ELSE
	bDone	:= FALSE;
END_IF

END_FUNCTION_BLOCK

// ---- POUs/METS/Common LIB/08_SOFTWARE LIB/Maths FBs/FB_CumulativeAverage.TcPOU
(* fAverage = sum of fInput samples / no of samples;  individual samples are not recorded *)
FUNCTION_BLOCK FB_CumulativeAverage
VAR_INPUT
	bEnable			: BOOL;		(* start cumulative calculation *)
	fInput			: LREAL;		(* input position *)
	tSamplePeriod	: TIME;		(* time period between each new value being logged *)
END_VAR
VAR_OUTPUT
	bRunning		: BOOL;		(* moving window being calculated without problem *)
	bNewValue		: BOOL;		(* set TRUE when a new value is logged and output is updated *)
	fAverage		: LREAL;	(* change in input value per second *)
	fMaxValue		: LREAL;	(* highest input value seen *)
	fMinValue		: LREAL;	(* lowest input value seen *)
END_VAR
VAR
	fbTaskTime		: FB_SYSTEM_TaskInfo;
	fTaskCycleTime	: LREAL;
	fbEnable		: R_TRIG;
	nLoggedSamples	: UDINT;
	fTimer			: LREAL;
	fSamplePeriod	: LREAL;
	fAccumulator	: LREAL;
END_VAR
(*
-------------------------------------------------------------------------------------------------
Date		Version	Author	Comments
-------------------------------------------------------------------------------------------------
30/01/2015	3.00.00	PB		LREAL now used in place of REAL

-------------------------------------------------------------------------------------------------
07/03/2012	1.09.00	PB		TaskTime calculated on rising edge of bEnable
05/02/2010	1.00.00	PB		Initial release

-------------------------------------------------------------------------------------------------
*)

(* detect rising edge of bEnable *)
fbEnable(CLK := bEnable);

(* generate average value *)
IF bEnable = TRUE THEN

	(* on rising edge of bEnable *)
	IF fbEnable.Q = TRUE THEN

		(* time base of current task *)
		fbTaskTime();
		fTaskCycleTime := fbTaskTime.fTaskTimeMicrosecs / 1000;

		fAccumulator := 0.0;
		nLoggedSamples := 0;
		fMaxValue := 0.0;
		fMinValue := 0.0;
	END_IF

	(* calculate sample period *)
	fSamplePeriod := MAX(fTaskCycleTime, TIME_TO_REAL(tSamplePeriod));

	(* update sample timer *)
	fTimer := fTimer + fTaskCycleTime;

	(* time to store new sample *)
	IF fTimer >= fSamplePeriod THEN

		(* set new value logged flag *)
		bNewValue := TRUE;

		(* update accumulator and samples and calculate new average *)
		fAccumulator := fAccumulator + fInput;
		nLoggedSamples := nLoggedSamples + 1;
		fAverage := F_SafeDIV(fAccumulator, UDINT_TO_REAL(nLoggedSamples));

		(* on 1st sample, set Max and Min Values = fInput *)
		IF nLoggedSamples = 1 THEN

			fMaxValue := fInput;
			fMinValue := fInput;
		END_IF

		(* update maximum and minimum values seen during average calculation *)
		fMaxValue := MAX(fInput, fMaxValue);
		fMinValue := MIN(fInput, fMinValue);

		(* remove complete sample time from timer *)
		fTimer := fTimer - fSamplePeriod;

	(* no new sample *)
	ELSE

		bNewValue := FALSE;
	END_IF

(* sampling disabled *)
ELSE

	bRunning := FALSE;
	bNewValue := FALSE;
	fAverage := fInput;
	nLoggedSamples := 0;
END_IF

END_FUNCTION_BLOCK

// ---- POUs/METS/Common LIB/08_SOFTWARE LIB/Maths FBs/FB_Interval.TcPOU
FUNCTION_BLOCK FB_Interval
(*
Version history:
Date		|	Version/Author 		|	Remark
----------------------------------------------------------------------------------------------------
04.07.12	|	2.000.001	PSA		|	Original Version
									|	Calculates the interval and ppm for 2 pulses.
*)
VAR_INPUT
	bSignal							: BOOL;						(* Input to detect the event *)
END_VAR
VAR_OUTPUT
	fInterval						: LREAL;					(* Gap between last 2 events  *)
	fPartsPerMinute					: LREAL;					(* Approximate parts per minute based on interval *)
END_VAR
VAR
	
	bInitOK 		: BOOL;
	fbTaskIndex		: GETCURTASKINDEX;
	
	fbSignalTrig					: R_TRIG;
	nCycleCount						: DWORD;
	nLastCycleCount					: DWORD;
END_VAR

fbSignalTrig(CLK := bSignal);

IF NOT bInitOK THEN
	(* get task indexc and task cycle time in seconds *)
	fbTaskIndex();
END_IF

bInitOK := fbTaskIndex.Index <> 0;

IF fbSignalTrig.Q AND bInitOK THEN
	
	nCycleCount :=  _TaskInfo[fbTaskIndex.Index].CycleCount;
	fInterval := DWORD_TO_LREAL(nCycleCount - nLastCycleCount) * (DWORD_TO_LREAL(_TaskInfo[fbTaskIndex.Index].CycleTime) / 10000000);
	nLastCycleCount :=  _TaskInfo[fbTaskIndex.Index].CycleCount;
	fPartsPerMinute := F_SafeDIV(60,fInterval);
END_IF

END_FUNCTION_BLOCK

// ---- POUs/METS/Common LIB/08_SOFTWARE LIB/Maths FBs/FB_MovingAverage.TcPOU
FUNCTION_BLOCK FB_MovingAverage
(*
Version history:
Date		|	Version/Author 		|	Remark
----------------------------------------------------------------------------------------------------
21.05.15	|	3.000.001	PSA		|	Original version
									|	Calculates a rolling average.
*)
VAR_INPUT
	bNewValue						: BOOL;						(* Input to detect the event *)
	bReset							: BOOL;						(* Resets the average value *)
	fLimit							: LREAL;					(* Limit value to inhibit bad data *)
END_VAR
VAR_OUTPUT
	nSamples						: DWORD := 1;
	fAverage						: LREAL := 0.0;
END_VAR
VAR
	fbTrig							: R_TRIG;
	fbResetTrig						: R_TRIG;
	FB_Interval1					: FB_Interval;
END_VAR

FB_Interval1(bSignal:= bNewValue);

fbTrig(CLK := bNewValue);
IF fbTrig.Q THEN
	IF FB_Interval1.fPartsPerMinute < fLimit THEN
		fAverage := ((fAverage * (nSamples - 1)) + FB_Interval1.fPartsPerMinute ) / nSamples;
		nSamples := nSamples + 1;
	END_IF
END_IF

fbResetTrig(CLK := bReset);
IF fbResetTrig.Q THEN
	nSamples := 1;
	fAverage := 0.0;
END_IF

END_FUNCTION_BLOCK

// ---- POUs/METS/Common LIB/08_SOFTWARE LIB/Maths FBs/FB_MovingAverageEvent.TcPOU
(* moving average over specified number if values logged on rising edge of bLogEvent *)
FUNCTION_BLOCK FB_MovingAverageEvent
VAR_INPUT
	bEnable			: BOOL;		(* set TRUE to enable moving average calculation.  fAverage = fInput when set FALSE *)
	bLogEvent		: BOOL;		(* log new value on FALSE-TRUE transition *)
	fInput			: LREAL;	(* input value *)
	nSamples		: UINT;		(* number of logged values to use *)
END_VAR
VAR_OUTPUT
	bRunning		: BOOL;		(* moving window being calculated without problem *)
	bError			: BOOL;		(* TRUE = nSamples is larger than size of internal array *)
	bNewValue		: BOOL;		(* set TRUE when a new value has been logged and fAverage updated *)
	fAverage		: LREAL;	(* moving average of last nSamples of fInput *)
	fMaxSample		: LREAL;	(* max value of samples being used *)
	fMinSample		: LREAL;	(* min value of samples being used *)
END_VAR
VAR
	fbEnable		: R_TRIG;
	arrValue		: ARRAY[1..120] OF LREAL;
	nMaxSamples		: UINT;
	fbLogEvent		: R_TRIG;
	nIndex			: UINT;
	nLoggedSamples	: UINT;
END_VAR
(*
-------------------------------------------------------------------------------------------------
Date		Version	Author	Comments
-------------------------------------------------------------------------------------------------
30/01/2015	3.00.00	PB		LREAL now used in place of REAL

-------------------------------------------------------------------------------------------------
07/03/2012	1.09.00	PB		MaxSamples is calculated and data array is cleared on rising edge of bEnable
05/02/2010	1.00.00	PB		Initial release

-------------------------------------------------------------------------------------------------
*)

(* detect rising edge of bEnable *)
fbEnable(CLK := bEnable);

(* log new value on rising edge of bExecute *)
fbLogEvent(CLK:= bLogEvent);

(* moving average enabled *)
IF bEnable = TRUE THEN

	(* on rising edge of bEnable *)
	IF fbEnable.Q = TRUE THEN

		(* clear array *)
		MEMSET(ADR(arrValue), 16#00, SIZEOF(arrValue));

		(* calculate max no of samples that can be handled *)
		nMaxSamples := SIZEOF(arrValue) / SIZEOF(arrValue[1]);
	END_IF

	(* no of samples specified exceeds size of array *)
	IF nSamples > nMaxSamples THEN

		(* set ERROR flag, use maximum number of samples allowed *)
		bError := TRUE;
		nSamples := nMaxSamples;
	END_IF

	(* log new value *)
	IF fbLogEvent.Q = TRUE THEN

		nLoggedSamples := MIN(nLoggedSamples + 1, nSamples);
		bNewValue := TRUE;

		(* shift data by 1 element in fValue and add new sample to fValue array *)
		MEMMOVE(ADR(arrValue[2]), ADR(arrValue[1]), SIZEOF(arrValue[1]) * (nMaxSamples - 1));
		arrValue[1] := fInput;

		(* calculate average value over specified period of time *)
		fAverage := 0.0;
		FOR nIndex := 1 TO nLoggedSamples DO

			(* add all sampled values *)
			fAverage := fAverage + arrValue[nIndex];

			(* new max sample or 1st value on scan *)
			IF arrValue[nIndex] > fMaxSample OR nIndex = 1 THEN

				fMaxSample := arrValue[nIndex];
			END_IF

			(* new min sample or 1st value on scan *)
			IF arrValue[nIndex] < fMinSample OR nIndex = 1 THEN

				fMinSample := arrValue[nIndex];
			END_IF
		END_FOR

		(* divide by number of samples used to return average value *)
		fAverage := F_SafeDIV(fAverage, UINT_TO_REAL(nLoggedSamples));

	(* no new value *)
	ELSE

		bNewValue := FALSE;
	END_IF

	bRunning := TRUE;

(* moving average disabled, output = input *)
ELSE

	bRunning := FALSE;
	bError := FALSE;
	bNewValue := FALSE;
	fAverage := fInput;
	nLoggedSamples := 0;
END_IF

END_FUNCTION_BLOCK

// ---- POUs/METS/Common LIB/08_SOFTWARE LIB/Maths FBs/FB_MovingAverageTimer.TcPOU
(* Returns a moving average over the last N cycles.  Values are taken on fixed timebase
and added to a buffer, new value replaces oldest value when 120 sample buffer is full. 
No of samples used for fAverage is calculated as tAveragePeriod / tSamplePeriod *)
FUNCTION_BLOCK FB_MovingAverageTimer
VAR_INPUT
	bEnable			: BOOL;		(* set TRUE to enable moving average calculation.  fAverage = fInput when set FALSE *)
	fInput			: LREAL;	(* input position *)
	tSamplePeriod	: TIME;		(* time period between each new value being logged, T#0ms = every cycle *)
	tAveragePeriod	: TIME;		(* time period over which to asses change of input value *)
END_VAR
VAR_OUTPUT
	bRunning		: BOOL;		(* moving window being calculated without problem *)
	bError			: BOOL;		(* error condition active *)
	bNewValue		: BOOL;		(* set TRUE when a new value is logged and output is updated *)
	fAverage		: LREAL;	(* change in input value per second *)
	fMaxSample		: LREAL;	(* max value of samples being used *)
	fMinSample		: LREAL;	(* min value of samples being used *)
END_VAR
VAR
	fbEnable		: R_TRIG;
	arrValue		: ARRAY[1..120] OF LREAL;
	fbTaskTime		: FB_SYSTEM_TaskInfo;
	fTaskCycleTime	: LREAL;
	nMaxSamples		: UINT;
	fSamplePeriod	: LREAL;
	fAveragePeriod	: LREAL;
	nSamples		: UINT;
	fTimer			: LREAL;
	nLoggedSamples	: UINT;
	nIndex			: UINT;
END_VAR
(*
-------------------------------------------------------------------------------------------------
Date		Version	Author	Comments
-------------------------------------------------------------------------------------------------
30/01/2015	3.00.00	PB		LREAL now used in place of REAL

-------------------------------------------------------------------------------------------------
07/03/2012	1.09.00	PB		TaskTime and MaxSamples are calculated and arrValue is cleared on rising edge of bEnable
05/02/2010	1.00.00	PB		Initial release

-------------------------------------------------------------------------------------------------
*)

(* detect rising edge of bEnable *)
fbEnable(CLK := bEnable);

(* moving average enabled *)
IF bEnable = TRUE THEN

	(* on rising edge of bEnable *)
	IF fbEnable.Q = TRUE THEN

		(* time base of current task *)
		fbTaskTime();
		fTaskCycleTime := fbTaskTime.fTaskTimeMicrosecs / 1000;

		(* clear array *)
		MEMSET(ADR(arrValue), 16#00, SIZEOF(arrValue));

		(* calculate max no of samples that can be handled *)
		nMaxSamples := SIZEOF(arrValue) / SIZEOF(arrValue[1]);
	END_IF

	(* calculate internal values required *)
	fSamplePeriod := MAX(fTaskCycleTime, TIME_TO_REAL(tSamplePeriod));
	fAveragePeriod := MAX(fTaskCycleTime, TIME_TO_REAL(tAveragePeriod));
	nSamples := lREAL_TO_UINT(F_SafeDIV(fAveragePeriod, fSamplePeriod));

	(* no of samples specified exceeds size of array *)
	IF nSamples > nMaxSamples THEN

		(* set ERROR flag, use maximum number of samples allowed *)
		bError := TRUE;
		nSamples := nMaxSamples;
	END_IF

	(* update timer *)
	fTimer := fTimer + fTaskCycleTime;

	(* time to store new sample *)
	IF fTimer >= fSamplePeriod THEN

		bNewValue := TRUE;
		nLoggedSamples := MIN(nLoggedSamples + 1, nSamples);

		(* shift data by 1 element in fValue and add new sample to array *)
		MEMMOVE(ADR(arrValue[2]), ADR(arrValue[1]), SIZEOF(arrValue[1]) * (nMaxSamples - 1));
		arrValue[1] := fInput;

		(* remove complete sample time from timer *)
		fTimer := fTimer - fSamplePeriod;

		(* calculate average value over specified period of time *)
		fAverage := 0.0;
		FOR nIndex := 1 TO nLoggedSamples DO

			(* add all sampled values *)
			fAverage := fAverage + arrValue[nIndex];

			(* new max sample or 1st value on scan *)
			IF arrValue[nIndex] > fMaxSample OR nIndex = 1 THEN

				fMaxSample := arrValue[nIndex];
			END_IF

			(* new min sample or 1st value on scan *)
			IF arrValue[nIndex] < fMinSample OR nIndex = 1 THEN

				fMinSample := arrValue[nIndex];
			END_IF
		END_FOR

		(* divide by number of samples used to return average value *)
		fAverage := F_SafeDIV(fAverage, UINT_TO_REAL(nLoggedSamples));

	(* no new sample *)
	ELSE

		bNewValue := FALSE;
	END_IF

	bRunning := TRUE;

(* moving average disabled *)
ELSE

	bRunning := FALSE;
	bError := FALSE;
	bNewValue := FALSE;
	fAverage := fInput;
	nLoggedSamples := 0;
END_IF

END_FUNCTION_BLOCK

// ---- POUs/METS/Common LIB/08_SOFTWARE LIB/Maths FBs/FB_MovingWindowEvent.TcPOU
(* Returns the difference between new value and historical value.
Values are added to a buffer on rising edge of bLogEvent, oldest value is deleted after 120 samples.
No of samples to be used is specified by nSamples *)
FUNCTION_BLOCK FB_MovingWindowEvent
VAR_INPUT
	bEnable			: BOOL;
	bLogEvent		: BOOL;		(* log new input value and time *)
	fInput			: LREAL;	(* input value *)
	fTime			: LREAL;	(* time in secs *)
	nSamples		: UINT;		(* number of events to log *)
END_VAR
VAR_OUTPUT
	bRunning		: BOOL;		(* moving window being calculated without problem *)
	bError			: BOOL;		(* error condition active *)
	bNewValue		: BOOL;		(* set TRUE when a new value is logged and output is updated *)
	fDeltaPerSec	: LREAL;	(* change in input value per second *)
	fDeltaPerMin	: LREAL;	(* change in input value per minute *)
	fDeltaPerHour	: LREAL;	(* change in input value per hour *)
END_VAR
VAR
	fbEnable		: R_TRIG;
	arrValue		: ARRAY[1..120] OF LREAL;
	arrTime			: ARRAY[1..120] OF LREAL;
	nMaxSamples		: UINT;
	nLoggedSamples	: UINT;
	fbLogEvent		: R_TRIG;
END_VAR
(*
-------------------------------------------------------------------------------------------------
Date		Version	Author	Comments
-------------------------------------------------------------------------------------------------
30/01/2015	3.00.00	PB		LREAL now used in place of REAL

-------------------------------------------------------------------------------------------------
07/03/2012	1.09.00	PB		MaxSamples is calculated and data arrays are cleared on rising edge of bEnable
05/02/2010	1.00.00	PB		Initial release

-------------------------------------------------------------------------------------------------
*)

(* detect rising edge of bEnable *)
fbEnable(CLK := bEnable);

(* check for rising edge on bLogEvent input *)
fbLogEvent(CLK:= bLogEvent);

(* moving window enabled *)
IF bEnable = TRUE THEN

	(* on rising edge of bEnable *)
	IF fbEnable.Q = TRUE THEN

		(* clear arrays *)
		MEMSET(ADR(arrValue), 16#00, SIZEOF(arrValue));
		MEMSET(ADR(arrTime), 16#00, SIZEOF(arrTime));

		(* calculate max no of samples that can be handled *)
		nMaxSamples := SIZEOF(arrValue) / SIZEOF(arrValue[1]);
	END_IF

	(* no of samples specified exceeds size of array *)
	IF nSamples > nMaxSamples THEN

		(* set ERROR flag, use maximum number of samples allowed *)
		bError := TRUE;
		nSamples := nMaxSamples;
	END_IF

	(* log new value *)
	IF fbLogEvent.Q = TRUE THEN

		bNewValue := TRUE;
		nLoggedSamples := MIN(nLoggedSamples + 1, nSamples);

		(* shift data by 1 element in fArray and add new sample to array *)
		MEMMOVE(ADR(arrValue[2]), ADR(arrValue[1]), SIZEOF(arrValue[1]) * (nMaxSamples - 1));
		MEMMOVE(ADR(arrTime[2]), ADR(arrTime[1]), SIZEOF(arrTime[1]) * (nMaxSamples - 1));
		arrValue[1] := fInput;
		arrTime[1] := fTime;

		(* need 2 samples before change of input over time can be calculated *)
		IF nLoggedSamples > 1 THEN

			(* calculate change of input over change of time *)
			fDeltaPerSec := F_SafeDIV((arrValue[1] - arrValue[nLoggedSamples]), (arrTime[1] - arrTime[nLoggedSamples]));
			fDeltaPerMin := fDeltaPerSec * 60.0;
			fDeltaPerHour := fDeltaPerMin * 60.0;
		END_IF

	(* no new sample *)
	ELSE

		bNewValue := FALSE;
	END_IF

(* moving window disabled *)
ELSE

	bRunning := FALSE;
	bError := FALSE;
	bNewValue := FALSE;
	fDeltaPerSec := 0.0;
	fDeltaPerMin := 0.0;
	nLoggedSamples := 0;
END_IF

END_FUNCTION_BLOCK

// ---- POUs/METS/Common LIB/08_SOFTWARE LIB/Maths FBs/FB_MovingWindowTimer.TcPOU
(* Returns the difference between new value and historical value.
Values are added to a buffer on a fixed timebase, oldest value is deleted after 120 samples.
Time difference between assessed values is specified by tWindowPeriod *)
FUNCTION_BLOCK FB_MovingWindowTimer
VAR_INPUT
	bEnable			: BOOL;
	fInput			: LREAL;	(* input position *)
	tSamplePeriod	: TIME;		(* time period between each new value being logged, T#0ms = every cycle *)
	tWindowPeriod	: TIME;		(* time period over which to asses change of input value *)
END_VAR
VAR_OUTPUT
	bRunning		: BOOL;		(* moving window being calculated without problem *)
	bError			: BOOL;		(* error condition active *)
	bNewValue		: BOOL;		(* set TRUE when a new value is logged and output is updated *)
	fDeltaPerSec	: LREAL;	(* change in input value per second *)
	fDeltaPerMin	: LREAL;	(* change in input value per minute *)
	fDeltaPerHour	: LREAL;	(* change in input value per hour *)
END_VAR
VAR
	fbEnable		: R_TRIG;
	fbTaskTime		: FB_SYSTEM_TaskInfo;
	fTaskCycleTime	: LREAL;
	arrValue		: ARRAY[1..120] OF LREAL;
	nMaxSamples		: UINT;
	fSamplePeriod	: LREAL;
	fWindowPeriod	: LREAL;
	nSamples		: UINT;
	fTimer			: LREAL;
	nLoggedSamples	: UINT;
END_VAR
(*
-------------------------------------------------------------------------------------------------
Date		Version	Author	Comments
-------------------------------------------------------------------------------------------------
30/01/2015	3.00.00	PB		LREAL now used in place of REAL

-------------------------------------------------------------------------------------------------
07/03/2012	1.09.00	PB		TaskTime and MaxSamples are calculated and arrValue is cleared on rising edge of bEnable
05/02/2010	1.00.00	PB		Initial release

-------------------------------------------------------------------------------------------------
*)

(* detect rising edge of bEnable *)
fbEnable(CLK := bEnable);

(* moving window enabled *)
IF bEnable = TRUE THEN

	(* on rising edge of bEnable *)
	IF fbEnable.Q = TRUE THEN

		(* time base of current task *)
		fbTaskTime();
		fTaskCycleTime := fbTaskTime.fTaskTimeMicrosecs / 1000;

		(* clear array *)
		MEMSET(ADR(arrValue), 16#00, SIZEOF(arrValue));

		(* calculate max no of samples that can be handled *)
		nMaxSamples := SIZEOF(arrValue) / SIZEOF(arrValue[1]);
	END_IF

	fSamplePeriod := MAX(fTaskCycleTime, TIME_TO_REAL(tSamplePeriod));
	fWindowPeriod := MAX(fTaskCycleTime, TIME_TO_REAL(tWindowPeriod));
	nSamples := lREAL_TO_UINT(F_SafeDIV(fWindowPeriod, fSamplePeriod));

	(* no of samples specified exceeds size of array *)
	IF nSamples > nMaxSamples THEN

		(* set ERROR flag, use maximum number of samples allowed *)
		bError := TRUE;
		nSamples := nMaxSamples;
	END_IF

	(* update timer *)
	fTimer := fTimer + fTaskCycleTime;

	(* time to store new sample *)
	IF fTimer >= fSamplePeriod THEN

		bNewValue := TRUE;
		nLoggedSamples := MIN(nLoggedSamples + 1, nSamples);

		(* shift data by 1 element in fArray and add new sample to array *)
		MEMMOVE(ADR(arrValue[2]), ADR(arrValue[1]), SIZEOF(arrValue[1]) * (nMaxSamples - 1));
		arrValue[1] := fInput;

		(* remove complete sample time from timer *)
		fTimer := fTimer - fSamplePeriod;

		(* calculate position change over specified number of samples *)
		fDeltaPerSec := F_SafeDIV((arrValue[1] - arrValue[nLoggedSamples]) * 1000.0, (fSamplePeriod * UINT_TO_REAL(nLoggedSamples)));
		fDeltaPerMin := fDeltaPerSec * 60.0;
		fDeltaPerHour := fDeltaPerMin * 60.0;

	(* no new sample *)
	ELSE

		bNewValue := FALSE;
	END_IF

(* moving window disabled *)
ELSE

	bRunning := FALSE;
	bError := FALSE;
	bNewValue := FALSE;
	fDeltaPerSec := 0.0;
	fDeltaPerMin := 0.0;
	nLoggedSamples := 0;
END_IF

END_FUNCTION_BLOCK

// ---- POUs/METS/Common LIB/08_SOFTWARE LIB/Maths FBs/F_ApplyTimeOffset.TcPOU
(* apply specified TIME offset to TIMESTRUCT value *)
FUNCTION F_ApplyTimeOffset : TIMESTRUCT
VAR_INPUT
	sTime			: TIMESTRUCT;	(* system time *)
	nTimeOffset		: DINT;			(* offset time, specified in ms *)
END_VAR
VAR
	nFileTime		: T_ULARGE_INTEGER;
END_VAR
(*
-------------------------------------------------------------------------------------------------
Date		Version	Author	Comments
-------------------------------------------------------------------------------------------------
30/01/2015	3.00.00	PB		Moved from Sewtec_CaseTrace.lib

-------------------------------------------------------------------------------------------------
03/08/2012	1.39.00	PB		Initial release

-------------------------------------------------------------------------------------------------
*)

(* offset time is specified *)
IF nTimeOffset <> 0 THEN

	(* convert TIMESTRUCT to T_ULARGE_INTEGER via T_FILETIME *)
	nFileTime := F_FileTimeToULarge(SYSTEMTIME_TO_FILETIME(sTime));

	(* positive time offset *)
	IF nTimeOffset >= 0 THEN

		(* convert DINT (1 = 1ms) to T_ULARGE_INTEGER (1 = 100ns) and add to system time *)
		nFileTime := UInt64Add64(nFileTime, UInt32x32To64(ABS(DINT_TO_DWORD(nTimeOffset)), 10000));

	(* negative time offset *)
	ELSE

		(* convert DINT (1 = 1ms) to T_ULARGE_INTEGER (1 = 100ns) and subtract from system time *)
		nFileTime := UInt64Sub64(nFileTime, UInt32x32To64(ABS(DINT_TO_DWORD(nTimeOffset)), 10000));
	END_IF

	(* convert T_ULARGE_INTEGER to TIMESTRUCT (via T_FILETIME *)
	F_ApplyTimeOffset := FILETIME_TO_SYSTEMTIME(F_ULargeToFileTime(nFileTime));

(* offset time = 0 *)
ELSE

	(* set Offset Time = System Time *)
	F_ApplyTimeOffset := sTime;
END_IF

END_FUNCTION

// ---- POUs/METS/Common LIB/08_SOFTWARE LIB/Maths FBs/F_ULargeToFileTime.TcPOU
(* convert value from 64-bit T_ULARGE_INTEGER to 64-bit T_FILETIME *)
FUNCTION F_ULargeToFileTime : T_FILETIME
VAR_INPUT
	nULarge			: T_ULARGE_INTEGER;
END_VAR
VAR
END_VAR
(*
-------------------------------------------------------------------------------------------------
Date		Version	Author	Comments
-------------------------------------------------------------------------------------------------
30/01/2015	3.00.00	PB		Moved from Sewtec_CaseTrace.lib

-------------------------------------------------------------------------------------------------
03/08/2012	1.39.00	PB		Initial release

-------------------------------------------------------------------------------------------------
*)

MEMMOVE(ADR(F_ULargeToFileTime), ADR(nULarge), SIZEOF(F_ULargeToFileTime));

END_FUNCTION

// ---- POUs/METS/Common LIB/08_SOFTWARE LIB/Maths FBs/F_CompareSign.TcPOU
(* F_CompareSign compares the sign of 2 LREAL values and gives TRUE if both values *)
(* are non-zero and have opposite sign *)
FUNCTION F_CompareSign : BOOL
VAR_INPUT
	fValue1		: LREAL;
	fValue2		: LREAL;
END_VAR
VAR
END_VAR
(*
-------------------------------------------------------------------------------------------------
Date		Version	Author	Comments
-------------------------------------------------------------------------------------------------
30/01/2015	3.00.00	PB		No change

-------------------------------------------------------------------------------------------------
05/02/10	1.00.00	PB		Initial release

-------------------------------------------------------------------------------------------------
*)

(* input values are both non-zero *)
IF fValue1 <> 0.0 AND fValue2 <> 0.0 THEN

	(* values have different signs *)
	IF F_GetSign(fValue1) <> F_GetSign(fValue2) THEN

		F_CompareSign := TRUE;

	(* values have same sign *)
	ELSE

		F_CompareSign := FALSE;
	END_IF

(* one of input values is zero *)
ELSE

	F_CompareSign := FALSE;
END_IF

END_FUNCTION

// ---- POUs/METS/Common LIB/08_SOFTWARE LIB/Maths FBs/F_GetSign.TcPOU
(* F_GetSign indicates the sign of the input LREAL value, set to 0 is input value is 0 *)
(* 1 = +ive, -1 = -ive *)
FUNCTION F_GetSign : INT
VAR_INPUT
	fValue		: LREAL;
END_VAR
VAR
END_VAR
(*
-------------------------------------------------------------------------------------------------
Date		Version	Author	Comments
-------------------------------------------------------------------------------------------------
30/01/2015	3.00.00	PB		No change

-------------------------------------------------------------------------------------------------
05/02/10	1.00.00	PB		Initial release

-------------------------------------------------------------------------------------------------
*)

(* input value is positive *)
IF fValue > 0.0 THEN

	F_GetSign := 1;

(* input value is negative *)
ELSIF fValue < 0.0 THEN

	F_GetSign := -1;

(* input value is zero *)
ELSE

	F_GetSign := 0;
END_IF

END_FUNCTION

// ---- POUs/METS/Common LIB/08_SOFTWARE LIB/Maths FBs/F_Interpolate.TcPOU
(* linear interpolation between 2 specified points (X,Y) using y=mx+c *)
FUNCTION F_Interpolate : LREAL
VAR_INPUT
	fX1			: LREAL;	(* X for defined point 1 *)
	fY1			: LREAL;	(* Y for defined point 1 *)
	fX2			: LREAL;	(* X for defined point 2 *)
	fY2			: LREAL;	(* Y for defined point 2 *)
	fCurrX		: LREAL;	(* current X value *)
END_VAR
VAR
END_VAR
(*
-------------------------------------------------------------------------------------------------
Date		Version	Author	Comments
-------------------------------------------------------------------------------------------------
30/01/2015	3.00.00	PB		Initial release

-------------------------------------------------------------------------------------------------
*)

(* X values are identical *)
IF fX2 = fX1 THEN

	(* graph is a vertical line and cannot interpolate, output is fixed *)
	F_Interpolate := fX1;

(* X values are different *)
ELSE

	(* apply linear interpolation *)
	F_Interpolate := (((fY2 - fY1) * (fCurrX - fX1)) / (fX2 - fX1)) + fY1;
END_IF

END_FUNCTION

// ---- POUs/METS/Common LIB/08_SOFTWARE LIB/Maths FBs/F_ModuloPos.TcPOU
(* converts absolute position to modulo position, 0 <= fModuloPos < fModuloFactor *)
FUNCTION F_ModuloPos : LREAL
VAR_INPUT
	fAbsPos			: LREAL;	(* absolute position *)
	fModuloFactor	: LREAL;	(* modulo factor *)
END_VAR
VAR
END_VAR
(*
-------------------------------------------------------------------------------------------------
Date		Version	Author	Comments
-------------------------------------------------------------------------------------------------
30/01/2015	3.00.00	PB		Initial release

-------------------------------------------------------------------------------------------------
*)

(* absolute position is +ive *)
IF fAbsPos >= 0 THEN

	(* LMOD produces modulo position *)
	F_ModuloPos := LMOD(fAbsPos, fModuloFactor);

(* absolute position is -ive *)
ELSE

	(* LMOD gives negative value, add fModuloFactor to convert to positive value *)
	F_ModuloPos := LMOD(fAbsPos, fModuloFactor) + fModuloFactor;
END_IF

END_FUNCTION

// ---- POUs/METS/Common LIB/08_SOFTWARE LIB/Memory FBs/FB_StructureMonitor.TcPOU
(* monitor memory area for change of data, max 64Kbytes *)
FUNCTION_BLOCK FB_StructureMonitor
VAR_INPUT
	bEnable			: BOOL;		(* set TRUE to enable monitoring *)
	pSourceData		: POINTER TO BYTE;	(* pointer to source data *)
	nSourceBytes	: UDINT;	(* no of data bytes *)
	tUpdateTime		: TIME;		(* update time *)
END_VAR
VAR_OUTPUT
	bDataChanged	: BOOL;		(* TRUE = data changed *)
	nTotalChanges	: UDINT;	(* total number of memory changes detected *)
END_VAR
VAR

	nCurrentCheckSum	: WORD;
	nLastCheckSum	: WORD;
	fbUpdateTimer		: FB_PulseGenerator;
END_VAR

(* update timer *)
fbUpdateTimer(
	bEnable		:= bEnable,
	tPeriod		:= tUpdateTime
);

(* data not changed on last pass *)
IF bDataChanged = FALSE THEN

	(* check for change of data *)
	IF fbUpdateTimer.bOutput = TRUE THEN

		nCurrentCheckSum := F_Checksum_CRC16(bEnable	:= bEnable, pSrcAddr := pSourceData, nBytes := nSourceBytes, nStartCRC := 16#FFFF);

		IF nCurrentCheckSum <> nLastCheckSum THEN

			nTotalChanges := nTotalChanges + 1;
			bDataChanged := TRUE;
		END_IF
	END_IF

(* data change detected on last pass *)
ELSE
	nLastCheckSum := nCurrentCheckSum;
	bDataChanged := FALSE;
END_IF

END_FUNCTION_BLOCK

// ---- POUs/METS/Common LIB/08_SOFTWARE LIB/Memory FBs/F_Checksum_CRC16.TcPOU
(* calculate 16-bit checksum on a memory area *)
FUNCTION F_Checksum_CRC16 : WORD
VAR_INPUT
	bEnable		: BOOL;				(* TRUE = calculate checksum *)
	pSrcAddr	: POINTER TO BYTE;	(* pointer to 1st byte of memory area *)
	nBytes		: UDINT;			(* no of bytes to be included in checksum calculation *)
	nStartCRC	: UINT;				(* initial value used for checksum calculation *)
END_VAR
VAR
END_VAR
(*
-------------------------------------------------------------------------------------------------
Date		Version	Author	Comments
-------------------------------------------------------------------------------------------------
30/01/2015	3.00.00	PB		No change

-------------------------------------------------------------------------------------------------
05/02/10	1.00.00	PB		Initial release

-------------------------------------------------------------------------------------------------
*)

(* calculate checksum when bEnable = TRUE *)
IF bEnable = TRUE THEN

	F_Checksum_CRC16 := F_DATA_TO_CRC16_CCITT(pSrcAddr, nBytes, nStartCRC);
END_IF

END_FUNCTION

// ---- POUs/METS/Common LIB/08_SOFTWARE LIB/Memory FBs/F_8BitsToByte.TcPOU
(* moves 8 bits into a single byte *)
FUNCTION F_8BitsToByte : BYTE
VAR_INPUT
	bInput1		: BOOL;
	bInput2		: BOOL;
	bInput3		: BOOL;
	bInput4		: BOOL;
	bInput5		: BOOL;
	bInput6		: BOOL;
	bInput7		: BOOL;
	bInput8		: BOOL;
END_VAR
VAR
END_VAR
(*
-------------------------------------------------------------------------------------------------
Date		Version	Author	Comments
-------------------------------------------------------------------------------------------------
30/01/2015	3.00.00	PB		Initial release

-------------------------------------------------------------------------------------------------
*)

F_8BitsToByte.0 := bInput1;
F_8BitsToByte.1 := bInput2;
F_8BitsToByte.2 := bInput3;
F_8BitsToByte.3 := bInput4;
F_8BitsToByte.4 := bInput5;
F_8BitsToByte.5 := bInput6;
F_8BitsToByte.6 := bInput7;
F_8BitsToByte.7 := bInput8;

END_FUNCTION

// ---- POUs/METS/Common LIB/08_SOFTWARE LIB/Memory FBs/F_GetBitState.TcPOU
(* returns status of specified bit from a DWORD value *)
FUNCTION F_GetBitState : BOOL
VAR_INPUT
	bEnable		: BOOL;		(* set TRUE to update output with state of target bit in nValue *)
	nTargetBit	: BYTE;		(* number of bit in nValue to be returned (0-31) *)
	nValue		: DWORD;	(* value from which target bit should be extracted *)
END_VAR
VAR
	nMaskValue	: DWORD;
END_VAR
(*
-------------------------------------------------------------------------------------------------
Date		Version	Author	Comments
-------------------------------------------------------------------------------------------------
30/01/2015	3.00.00	PB		No change

-------------------------------------------------------------------------------------------------
21/05/2010	1.03.00	PB		Initial release

-------------------------------------------------------------------------------------------------
*)

(* bit evaluation is enabled *)
IF bEnable = TRUE THEN

	(* target bit must be 0-31 *)
	IF nTargetBit <= 31 THEN

		(* calculate mask value from specified target bit *)
		nMaskValue := lREAL_TO_DWORD(EXPT(2, nTargetBit));

		(* compare nDWord AND nMaskValue, target bit is TRUE if value > 0 *)
		IF (nValue AND nMaskValue) > 0 THEN

			F_GetBitState := TRUE;

		(* target bit is FALSE *)
		ELSE

			F_GetBitState := FALSE;
		END_IF

	(* target bit out of range *)
	ELSE

		F_GetBitState := FALSE;
	END_IF

(* bit evaluation disabled *)
ELSE

	F_GetBitState := FALSE;
END_IF

END_FUNCTION

// ---- POUs/METS/Common LIB/08_SOFTWARE LIB/Memory FBs/F_PointerToByteADD.TcPOU
(* add offset to POINTER TO BYTE value *)
FUNCTION F_PointerToByteADD : PVOID
VAR_INPUT
	pPointer		: PVOID;	(* base pointer *)
	nOffset			: UDINT;			(* pointer offset *)
END_VAR
VAR
	nPointer		: ULINT;
	nPointerOffset	: ULINT;
END_VAR
(*
-------------------------------------------------------------------------------------------------
Date		Version	Author	Comments
-------------------------------------------------------------------------------------------------
30/01/2015	3.00.00	PB		No change

-------------------------------------------------------------------------------------------------
05/02/10	1.00.00	PB		Initial release

-------------------------------------------------------------------------------------------------
*)

nPointer := pPointer;					(* convert pointer to UDINT *)
nPointerOffset := nPointer + nOffset;	(* add offset *)
F_PointerToByteADD := nPointerOffset;	(* convert UDINT back to pointer *)

END_FUNCTION

// ---- POUs/METS/Common LIB/08_SOFTWARE LIB/Memory FBs/F_PointerToWordADD.TcPOU
(* add offset to POINTER TO WORD value *)
FUNCTION F_PointerToWordADD : PVOID
VAR_INPUT
	pPointer		: PVOID;	(* base pointer *)
	nOffset			: UDINT;			(* pointer offset *)
END_VAR
VAR
	nPointer		: ULINT;
	nPointerOffset	: ULINT;
END_VAR
(*
-------------------------------------------------------------------------------------------------
Date		Version	Author	Comments
-------------------------------------------------------------------------------------------------
30/01/2015	3.00.00	PB		No change

-------------------------------------------------------------------------------------------------
05/02/10	1.00.00	PB		Initial release

-------------------------------------------------------------------------------------------------
*)

nPointer := pPointer;					(* convert pointer to UDINT *)
nPointerOffset := nPointer + nOffset;	(* add offset *)
F_PointerToWordADD := nPointerOffset;	(* convert UDINT back to pointer *)

END_FUNCTION

// ---- POUs/METS/Common LIB/08_SOFTWARE LIB/Memory FBs/F_SetBitState.TcPOU
(* updates state of specified bit in nDWord value *)
FUNCTION F_SetBitState : DWORD
VAR_INPUT
	bEnable		: BOOL;		(* set TRUE to update state of target bit in nValue *)
	nTargetBit	: BYTE;		(* bit number of bit to be updated (0-31) *)
	nSetState	: BOOL;		(* state to which nTargetBit should be set *)
END_VAR

VAR
	nMaskValue	: DWORD;
END_VAR
(*
-------------------------------------------------------------------------------------------------
Date		Version	Author	Comments
-------------------------------------------------------------------------------------------------
30/01/2015	3.00.00	PB		No change

-------------------------------------------------------------------------------------------------
26/05/2010	1.03.01	PB		nValue now updated as well as F_SetBitState
21/05/2010	1.03.00	PB		Initial release

-------------------------------------------------------------------------------------------------
*)
(*All VAR_IN_OUT variables have been moved to the end of the declaration due to compatibility reasons*)
VAR_IN_OUT
	nValue		: DWORD;	(* value in which target bit should be updated *)
END_VAR

(* bit update is enabled *)
IF bEnable = TRUE THEN

	(* target bit must be 0-31 *)
	IF nTargetBit <= 31 THEN

		(* calculate mask value from specified target bit *)
		nMaskValue := LREAL_TO_DWORD(EXPT(2, nTargetBit));

		nValue := (nValue AND NOT nMaskValue) + (BOOL_TO_DWORD(nSetState) * nMaskValue);

	(* target bit out of range *)
	ELSE

		nValue := nValue;
	END_IF

(* bit update disabled *)
ELSE

	nValue := nValue;
END_IF

F_SetBitState := nValue;

END_FUNCTION

// ---- POUs/METS/Common LIB/08_SOFTWARE LIB/String FBs/FB_ExtractLongString.TcPOU
(* extracts a sub-string defined by prefix and suffix *)
FUNCTION_BLOCK FB_ExtractLongString
VAR_INPUT
	bExtractData		: BOOL;			(* set TRUE to remove prefix and suffix from strData *)
	nExtractChars		: UINT;			(* if suffix is blank, number of data chars to extract *)
	strPrefix			: T_MaxString;	(* prefix string *)
	strSuffix			: T_MaxString;	(* suffix string *)
END_VAR
VAR_IN_OUT
	strString			: T_LongSTRING;	(* string to be searched *)
END_VAR
VAR_OUTPUT
	bStringFound		: BOOL;			(* TRUE = sub-string with matching prefix/suffix found *)
	nStartPos			: UINT;			(* start pos of extracted string in strString *)
	strData				: T_LongSTRING;	(* extracted data *)
END_VAR
VAR
	nStringLen			: UINT;
	nPrefixLen			: UINT;
	nSuffixLen			: UINT;
	nEndPos				: UINT;
	bStartPosFound		: BOOL;
	bEndPosFound		: BOOL;
	nChars				: UINT;
	nMaxIndex			: UINT;
	nIndex				: UINT;

END_VAR
(*
-------------------------------------------------------------------------------------------------
DATE		Version	Author	Comments
-------------------------------------------------------------------------------------------------
30/01/2015	3.00.00	PB		Initial release

-------------------------------------------------------------------------------------------------
*)

(* calc string lengths *)
nStringLen := UDINT_TO_UINT(LEN2(ADR(strString)));
nPrefixLen := INT_TO_UINT(LEN(strPrefix));
nSuffixLen := INT_TO_UINT(LEN(strSuffix));

(* string to be searched is not empty and prefix or suffix or no or chars to extract is defined *)
IF nStringLen > 0 AND (nPrefixLen > 0 OR nSuffixLen > 0 OR nExtractChars > 0) THEN

	(* clear outputs *)
	bStringFound := FALSE;
	nChars := 0;
	nStartPos := 0;
	strData := '';

	(* initialise char index values *)
	bStartPosFound := FALSE;
	bEndPosFound := FALSE;
	nEndPos := 0;

	(* max search index, based on string length - 1 due to starting at 0 and length of prefix *)
	nMaxIndex := (nStringLen - 1) + (nPrefixLen - 1);

	(* for each character in the string *)
	FOR nIndex := 0 TO nMaxIndex DO

		(*IF nIndex = nMaxIndex  AND NOT bStartPosFound THEN

			strString :='1';

		(* prefix has not been found *)
		ELS*)IF bStartPosFound = FALSE THEN

			(* no prefix defined  *)
			IF nPrefixLen = 0 THEN

				(* start at beginning if string *)
				nStartPos := 1;
				bStartPosFound := TRUE;

			(* prefix defined  *)
			ELSE

				(* compare partial string with prefix *)
				IF MEMCMP(ADR(strString) + nIndex, ADR(strPrefix), nPrefixLen) = 0 THEN

					(* prefix position found *)
					nStartPos := nIndex + 1;
					bStartPosFound := TRUE;

					(* skip to end of prefix to continue search *)
					nIndex := nIndex + nPrefixLen - 1;
				END_IF
			END_IF

		(* suffix has not been found *)
		ELSIF bEndPosFound = FALSE THEN

			(* no suffix defined  *)
			IF nSuffixLen = 0 THEN

				(* start at 1st char of string *)
				bEndPosFound := TRUE;

				(* calculate end position *)
				nEndPos := MIN((nStartPos - 1) + nExtractChars + nPrefixLen, nStringLen);

			(* suffix defined  *)
			ELSE

				(* compare partial string with suffix *)
				IF MEMCMP(ADR(strString) + nIndex, ADR(strSuffix), nSuffixLen) = 0 THEN

					(* suffix position found, calculate end position *)
					nEndPos := nIndex + nSuffixLen;
					bEndPosFound := TRUE;

					(* no prefix defined and number of chars to extract is defined *)
					IF nPrefixLen = 0 AND nExtractChars > 0 THEN

						(* re-calculate start position *)
						nStartPos := MAX(nEndPos - nExtractChars - 1, 1);
					END_IF

					(* search complete, quit FOR loop *)
					EXIT;
				END_IF
			END_IF

		(* prefix and suffix found *)
		ELSE

			(* quit FOR loop *)
			EXIT;
		END_IF
	END_FOR

	(* start and end positions known *)
	IF bStartPosFound = TRUE AND bEndPosFound = TRUE THEN

		(* string has been found *)
		bStringFound := TRUE;

		(* return string without prefix and suffix *)
		IF bExtractData = TRUE THEN

			(* total chars to be moved to strData *)
			nChars := (nEndPos - (nStartPos - 1)) - nPrefixLen - nSuffixLen;

			(* 1 or more chars to be moved *)
			IF nChars > 0 THEN

				(* move data to strData *)
				MEMMOVE(ADR(strData), ADR(strString) + (nStartPos - 1) + nPrefixLen, nChars);
			END_IF

		(* return string with prefix and suffix *)
		ELSE

			(* total chars to be moved to strData *)
			nChars := nEndPos - (nStartPos - 1);

			(* 1 or more chars to be moved *)
			IF nChars > 0 THEN

				(* move data to strData *)
				MEMMOVE(ADR(strData), ADR(strString) + (nStartPos - 1), nChars);
			END_IF
		END_IF

		(* terminate strData *)
		MEMSET(ADR(strData) + nChars, 16#00, 1);

		(* 1 or more chars after strSuffix *)
		IF nStringLen > (nEndPos - (nStartPos - 1)) THEN

			(* shift post-suffix chars to prefix position *)
			MEMMOVE(ADR(strString) + (nStartPos - 1), ADR(strString) + nEndPos, nStringLen - (nEndPos - (nStartPos - 1)));
		END_IF

		(* terminate strString *)
		MEMSET(ADR(strString) + nStringLen - (nEndPos - (nStartPos - 1)), 16#00, 1);
	END_IF

(* string to be searched is empty or prefix and suffix and both blank *)
ELSE

	(* clear outputs *)
	bStringFound := FALSE;
	nChars := 0;
	strData := '';
END_IF

END_FUNCTION_BLOCK

// ---- POUs/METS/Common LIB/08_SOFTWARE LIB/String FBs/FB_ExtractString_v2.TcPOU
(* extracts a sub-string defined by prefix and suffix *)
FUNCTION_BLOCK FB_ExtractString_v2
VAR_INPUT
	bIgnoreCase		: BOOL;
	strPrefix		: STRING(10);	(* prefix string *)
	strSuffix		: STRING(10);	(* suffix string *)
	nExtractChars	: BYTE;			(* if suffix is blank, >0 = no of chars to extract , 0 = remainder of string *)
END_VAR
VAR_IN_OUT
	strString		: T_MaxString;	(* string to be searched *)
END_VAR
VAR_OUTPUT
	bStringFound	: BOOL;			(* TRUE = sub-string with matching prefix/suffix found *)
	nChars			: INT;			(* no of chars in sub-string *)
	strResult		: T_MaxString;	(* sub-string with prefix and suffix *)
END_VAR
VAR
	nPrefixPos		: INT;
	nSuffixPos		: INT;
	nIndex			: INT;
	strStringInt	: T_MaxString;
	strPrefixInt	: STRING(10);
	strSuffixInt	: STRING(10);
	strCheckString	: STRING(10);
END_VAR
(*
-------------------------------------------------------------------------------------------------
DATE		Version	Author	Comments
-------------------------------------------------------------------------------------------------
06/07/2011	1.23.00	PB		Pre-check added to ensure that strString is not empty.
07/06/2011	1.19.00	PB		bIgnoreCase input added, set to TRUE to ignore upper/lower case when matching Prefix and Suffix.
31/01/2011	1.08.03	PB		Bug fix - strings now handled correctly if strSuffix is longer than 1 char.
							Search for suffix changed to start after prefix position.
22/11/2010	1.07.01	PB		Initial release.

-------------------------------------------------------------------------------------------------
*)

(* string to be searched is not empty *)
IF LEN(strString) > 0 THEN

	(* matching for Prefix and Suffix is case-sesnsitive *)
	IF bIgnoreCase = FALSE THEN

		(* internal comparators are not changed *)
		strStringInt := strString;
		strPrefixInt := strPrefix;
		strSuffixInt := strsuffix;

	(* ignore case when matching for Prefix and Suffix *)
	ELSE

		(* internal comparators are all converted to lower case *)
		strStringInt := F_ToLCase(strString);
		strPrefixInt := F_ToLCase(strPrefix);
		strSuffixInt := F_ToLCase(strsuffix);
	END_IF

	(* prefix is blank *)
	IF strPrefixInt = '' THEN

		(* start at beginning of string *)
		nPrefixPos := 1;

	(* prefix is not blank *)
	ELSE

		(* find 1st occurrence of prefix in strString *)
		nPrefixPos := FIND(strStringInt, strPrefixInt);
	END_IF

	(* suffix is blank *)
	IF strSuffixInt = '' THEN
	
		(* no of chars not specified *)
		IF nExtractChars = 0 THEN
	
			(* finish at end of string *)
			nSuffixPos := LEN(strStringInt);
	
		(* no of chars specified *)
		ELSE
	
			(* finish at end of string *)
			nSuffixPos := nPrefixPos + nExtractChars - 1;
		END_IF
	
	(* suffix is not blank *)
	ELSE
	
		nSuffixPos := 0;
	
		(* find 1st occurrence of suffix in strString AFTER position of strPrefix *)
		FOR nIndex := nPrefixPos + LEN(strPrefixInt) TO LEN(strStringInt) DO
	
			(* extract string same length as suffix string *)
			strCheckString := MID(strStringInt, LEN(strSuffixInt), nIndex);
	
			(* extracted string = suffix string *)
			IF strCheckString = strSuffixInt THEN
	
				(* position of suffix string *)
				nSuffixPos := nIndex;
				EXIT;
			END_IF
		END_FOR
	END_IF
	
	
	(* prefix and suffix both exist *)
	IF nPrefixPos > 0 AND nSuffixPos > 0 THEN
	
		(* extract sub-string *)
		strResult := MID(strString, nSuffixPos + MAX(LEN(strSuffixInt), 1) - nPrefixPos, nPrefixPos);

		(* delete sub-string *)
		strString := DELETE(strString, nSuffixPos + MAX(LEN(strSuffixInt), 1) - nPrefixPos, nPrefixPos);
	
		(* update outputs *)
		bStringFound := TRUE;
		nChars := LEN(strResult);
	
	(* no prefix or suffix defined, cannot search for string *)
	ELSE
	
		strResult := '';
		bStringFound := FALSE;
		nChars := 0;
	END_IF

(* string to be searched is empty *)
ELSE

	(* reset outputs *)
	bStringFound := FALSE;
	nChars := 0;
	strResult := '';
END_IF

END_FUNCTION_BLOCK

// ---- POUs/METS/Common LIB/08_SOFTWARE LIB/String FBs/F_AddPadding.TcPOU
FUNCTION F_AddPadding : STRING
VAR_INPUT
	nNumber:		INT;
	nSize:			UINT;
END_VAR
VAR
	sTemp: STRING;
END_VAR

sTemp := INT_TO_STRING(nNumber);

WHILE LEN(sTemp) < nSize DO
	sTemp := CONCAT('0',sTemp);
END_WHILE

F_AddPadding := sTemp;

END_FUNCTION

// ---- POUs/METS/Common LIB/08_SOFTWARE LIB/String FBs/F_AddPaddingUDINT.TcPOU
FUNCTION F_AddPaddingUDINT : STRING
VAR_INPUT
	nNumber:		UDINT;
	nSize:			UINT;
END_VAR
VAR
	sTemp: STRING;
END_VAR

sTemp := UDINT_TO_STRING(nNumber);

WHILE LEN(sTemp) < nSize DO
	sTemp := CONCAT('0',sTemp);
END_WHILE

F_AddPaddingUDINT := sTemp;

END_FUNCTION

// ---- POUs/METS/Common LIB/08_SOFTWARE LIB/String FBs/F_IsNumber.TcPOU
FUNCTION F_IsNumber : BOOL
(*Returns true if the charachter is a number*)
VAR_INPUT
	sChr				: STRING(1);
END_VAR
VAR
END_VAR

F_IsNumber := (F_ToASC(sChr) >= 16#30 AND F_ToASC(sChr) <= 16#39);

END_FUNCTION

// ---- POUs/METS/Common LIB/08_SOFTWARE LIB/String FBs/F_StringAddSuffix.TcPOU
(* add specified char(s) to the end of a string to make up to specified length *)
FUNCTION F_StringAddSuffix : T_MaxString
VAR_INPUT
	sString		: T_MaxString;	(* initial string *)
	nTargetLen 		: UINT;			(* string length required *)
	sChar			: STRING(1);	(* char to be appended to string *)
END_VAR
VAR
	nStringLen		: UINT;
	nCharsReq		: UINT;
END_VAR
(*
-------------------------------------------------------------------------------------------------
Date		Version	Author	Comments
-------------------------------------------------------------------------------------------------
30/01/2015	3.00.00	PB		Initial release

-------------------------------------------------------------------------------------------------
*)

(* length of input string *)
nStringLen := TO_UINT(LEN(sString));

(* Chekck target string is longer than processing string *)
IF nTargetLen >= nStringLen THEN
	
	(* total suffix chars required *)
	nCharsReq := MIN(nTargetLen, SIZEOF(F_StringAddSuffix) - 1) - nStringLen;
	
	(* string needs additional chars *)
	IF nCharsReq > 0 THEN
	
		(* append strString to output string *)
		MEMMOVE(ADR(F_StringAddSuffix), ADR(sString), nStringLen);
	
		(* set suffix chars to specified character *)
		MEMSET(ADR(F_StringAddSuffix) + nStringLen, F_ToASC(sChar), nCharsReq);
	
		(* reset last char to 16#00 to terminate the string *)
		MEMSET(ADR(F_StringAddSuffix) + nStringLen + nCharsReq, 16#00, 1);
	
	(* no additional chars required *)
	ELSE
	
		(* copy strString to output *)
		F_StringAddSuffix := sString;
	END_IF
ELSE
	(* copy shrinced strString to output *)
	F_StringAddSuffix := LEFT(sString, TO_INT(nTargetLen));
END_IF

END_FUNCTION

// ---- POUs/METS/Common LIB/08_SOFTWARE LIB/String FBs/F_ValidateString.TcPOU
(* checks a string for various characteristics and returns a string if validation fails *)
FUNCTION F_ValidateString : T_MaxString
VAR_INPUT
	strFieldData		: T_MaxString;	(* string to be examined *)
	nExpectedChars		: BYTE;			(* >0 = no of chars expected in string, 0 = chars not counted but string must not be empty *)
	nMaxChars			: UINT;			(* >0 = max no of chars allowed in strFieldData, 0 = do not check *)
	bNumCharsOnly		: BOOL;			(* TRUE = all chars are checked to ensure only numerical (0-9) chars are present *)
	bDecPointAllowed	: BOOL;			(* TRUE = decimal point is allowed in a numerical string *)
END_VAR
VAR
	nIndex				: INT;
	nCharValue			: BYTE;
END_VAR
(*
-------------------------------------------------------------------------------------------------
DATE		Version	Author	Comments
-------------------------------------------------------------------------------------------------
30/01/2015	3.00.00	PB		Initial release

-------------------------------------------------------------------------------------------------
*)

(* string contains data *)
IF LEN(strFieldData) > 0 THEN

	(* field data length exceeds specified maximum no of chars *)
	IF nMaxChars > 0 AND LEN(strFieldData) >= nMaxChars THEN

		F_ValidateString := 'XML field data contains too many chars';

	(* string has expected no of chars OR string length does not matter *)
	ELSIF LEN(strFieldData) = nExpectedChars OR nExpectedChars = 0 THEN

		(* string must only have numerical chars *)
		IF bNumCharsOnly = TRUE THEN

			(* check each char in the string *)
			FOR nIndex := 1 TO LEN(strFieldData) DO

				(* convert char to ASCII value *)
				nCharValue := F_ToASC(MID(strFieldData, 1, nIndex));

				(* string char is valid if 0-9, decimal point also allowed if enabled *)
				IF (nCharValue >= F_ToASC('0') AND nCharValue <= F_ToASC('9')) OR (nCharValue = F_ToASC('.') AND bDecPointAllowed = TRUE) THEN

					F_ValidateString := '';

				(* invalid char *)
				ELSE

					F_ValidateString := F_CONCAT3('Invalid char "', MID(strFieldData, 1, nIndex), '" found');
					EXIT;
				END_IF
			END_FOR

		(* string can be alpha-numeric chars *)
		ELSE

			F_ValidateString := '';
		END_IF

	(* string has incorrect no of chars *)
	ELSE

		F_ValidateString := F_CONCAT4('Expected length = ', BYTE_TO_STRING(nExpectedChars), ', actual length = ', INT_TO_STRING(LEN(strFieldData)));
	END_IF

(* empty string *)
ELSE

	F_ValidateString := 'Empty';
END_IF

END_FUNCTION

// ---- POUs/METS/Common LIB/08_SOFTWARE LIB/String FBs/F_ValidateString_Code.TcPOU
(* checks a string for various characteristics and returns a code if validation fails *)
FUNCTION F_ValidateString_Code : UDINT
VAR_INPUT
	strFieldData		: T_MaxString;	(* string to be examined *)
	nExpectedChars		: BYTE;			(* >0 = no of chars expected in string, 0 = chars not counted but string must not be empty *)
	nMaxChars			: UINT;			(* >0 = max no of chars allowed in strFieldData, 0 = do not check *)
	bNumCharsOnly		: BOOL;			(* TRUE = all chars are checked to ensure only numerical (0-9) chars are present *)
	bDecPointAllowed	: BOOL;			(* TRUE = decimal point is allowed in a numerical string *)
END_VAR
VAR
	nIndex				: INT;
	nCharValue			: BYTE;
END_VAR
(*
-------------------------------------------------------------------------------------------------
DATE		Version	Author	Comments
-------------------------------------------------------------------------------------------------
30/01/2015	3.00.00	PB		Initial release

-------------------------------------------------------------------------------------------------
*)

(* string contains data *)
IF LEN(strFieldData) > 0 THEN

	(* field data length exceeds specified maximum no of chars *)
	IF nMaxChars > 0 AND LEN(strFieldData) > nMaxChars THEN

		F_ValidateString_Code := 6;

	(* string has expected no of chars OR string length does not matter *)
	ELSIF LEN(strFieldData) = nExpectedChars OR nExpectedChars = 0 THEN

		(* string must only have numerical chars *)
		IF bNumCharsOnly = TRUE THEN

			(* check each char in the string *)
			FOR nIndex := 1 TO LEN(strFieldData) DO

				(* convert char to ASCII value *)
(*				nCharValue := ASC(MID(strFieldData, 1, nIndex));*)
				nCharValue := F_ToASC(MID(strFieldData, 1, nIndex));

				(* string char is valid if 0-9, decimal point also allowed if enabled *)
				IF (nCharValue >= F_ToASC('0') AND nCharValue <= F_ToASC('9')) OR (nCharValue = F_ToASC('.') AND bDecPointAllowed = TRUE) THEN

					F_ValidateString_Code := 0;

				(* decimal point found but not allowed *)
				ELSIF nCharValue = F_ToASC('.') AND bDecPointAllowed = FALSE THEN

					F_ValidateString_Code := 5;
					EXIT;

				(* other invalid char found *)
				ELSE

					F_ValidateString_Code := 4;
					EXIT;
				END_IF
			END_FOR

		(* string can be alpha-numeric chars *)
		ELSE

			F_ValidateString_Code := 0;
		END_IF

	(* string is too short *)
	ELSIF LEN(strFieldData) < nExpectedChars THEN

		F_ValidateString_Code := 2;

	(* string is too long *)
	ELSIF LEN(strFieldData) > nExpectedChars THEN

		F_ValidateString_Code := 3;
	END_IF

(* empty string *)
ELSE

	F_ValidateString_Code := 1;
END_IF

END_FUNCTION

// ---- POUs/METS/Common LIB/08_SOFTWARE LIB/String FBs/F_WriteEscapeCharacters.TcPOU
FUNCTION F_WriteEscapeCharacters : T_MaxString
VAR_INPUT
	Value		: T_MaxString;
END_VAR
VAR
	nPosition	: INT;
END_VAR

nPosition := FIND(Value, '&');
IF nPosition > 0 THEN

	F_WriteEscapeCharacters := REPLACE(Value, '&amp;',1 , nPosition);

(*	F_WriteEscapeCharacters := LEFT(Value, nPosition - 1);
	F_WriteEscapeCharacters := CONCAT(F_WriteEscapeCharacters, '&amp;');
	F_WriteEscapeCharacters :=  CONCAT(F_WriteEscapeCharacters, RIGHT(Value, LEN(Value) - (nPosition)));
*)
ELSE

	F_WriteEscapeCharacters := Value;

END_IF

END_FUNCTION

// ---- POUs/METS/Common LIB/08_SOFTWARE LIB/String FBs/F_ZeroPadString.TcPOU
(* append leading zeroes to a string to make up to specified length, max 19 chars *)
FUNCTION F_ZeroPadString : STRING(19)
VAR_INPUT
	strString		: STRING(19);	(* initial string *)
	nPadLength 		: BYTE;		(* string length required *)
END_VAR
VAR
	nMaxLength		: BYTE;
END_VAR
(*
-------------------------------------------------------------------------------------------------
Date		Version	Author	Comments
-------------------------------------------------------------------------------------------------
03/08/2012	1.39.00	PB		String lengths reduced to 19 characters.
							Trap added to prevent PLC from crashing if nPadLength > 19.
12/11/2010	1.07.00	PB		Initial release

-------------------------------------------------------------------------------------------------
*)

(* max string length *)
nMaxLength := SIZEOF(F_ZeroPadString) - 1;

(* initial string *)
F_ZeroPadString := strString;

(* string length is shorter than required/max length *)
WHILE LEN(F_ZeroPadString) < MIN(nPadLength, nMaxLength) DO

	(* append leading '0' char to string *)
	F_ZeroPadString := CONCAT('0', F_ZeroPadString);
END_WHILE

END_FUNCTION

// ---- POUs/METS/Common LIB/08_SOFTWARE LIB/TCP FBs/FB_TCP_ClientPortCtrl.TcPOU
(* TCP port ctrl and monitoring for Client-Server devices *)
FUNCTION_BLOCK FB_TCP_ClientPortCtrl
VAR_INPUT
	bEnable				: BOOL;			(* set TRUE to enable TCP connection *)
	strRemoteIPAddr		: T_IPv4Addr;	(* IP address for remote device *)
	nRemotePortNo		: UINT;			(* port number for remote device *)
	tReconnectTime		: TIME;			(* TCP reconnect time *)
END_VAR
VAR_OUTPUT
	bConnected			: BOOL;			(* TRUE = TCP port is currently open *)
	bError				: BOOL;			(* TRUE = error occurred when opening TCP port *)
	nErrorID			: UDINT;		(* TRUE = error code *)
	hSocket				: T_HSocket;	(* TCP socket handle *)
	nSyncOffset			: DINT;			(* sync offset value to spread TCP Server access load *)
	eSocketState		: E_SocketConnectionState;	(* TCP socket state *)
END_VAR
VAR
	eTCPState			: E_TCPIP_State;
	strTargetIPAddr		: T_IPv4Addr;
	arrTargetIPAddr		: T_IPv4AddrArr;
	nTargetPortNo		: UDINT;
	fbTCPPortCtrl		: FB_ClientServerConnection;
END_VAR
(*
-------------------------------------------------------------------------------------------------
Date		Version	Author	Comments
-------------------------------------------------------------------------------------------------
30/01/2015	3.00.00	PB		No change

-------------------------------------------------------------------------------------------------
16/08/2012	1.40.02	PB		TCP status check now disabled if tStatusTime = T#0ms
							TCP status now check on rising edge of bEnable and every specified tStatusTime
							FB now re-connects properly if strRemoteIPAddr or nRemotePortNo are changed while TCP connection is active
							bError and nErrorID now linked directly to FB_ClientServerConnection, solves problem of auto-recovery due to incorrect status reporting.
26/01/2012	1.37.01	PB		Brackets added to ensure logic condition for when TCP connection can be disconnected is clear
22/11/2011	1.34.00	PB		tReconnectTime input added
17/11/2011	1.33.00	PB		Initial release

-------------------------------------------------------------------------------------------------
*)

CASE eTCPState OF

	(* TCP connetion not active *)
	E_TCPIP_IDLE:

		(* TCP connection is enabled *)
		IF bEnable = TRUE THEN

			(* target IP address and port number *)
			strTargetIPAddr := strRemoteIPAddr;
			nTargetPortNo := nRemotePortNo;

			(* convert target IP address to bytes *)
			arrTargetIPAddr := F_ScanIPv4AddrIds(strTargetIPAddr);
			nSyncOffset := arrTargetIPAddr[3] MOD 10;

			eTCPState := E_TCPIP_CONNECT;
		END_IF


	(* open TCP connection *)
	E_TCPIP_CONNECT:

		(* TCP connection not required or status check not active *)
		IF bEnable = FALSE (*OR (bConnect = FALSE AND bCheckStatus = FALSE)*) THEN

			eTCPState := E_TCPIP_DISCONNECT;

		(* TCP connect error or remote IP address or port number have changed while connection is active *)
		ELSIF fbTCPPortCtrl.bError = TRUE OR (strRemoteIPAddr <> strTargetIPAddr AND strTargetIPAddr <> '') OR (nRemotePortNo <> nTargetPortNo AND nTargetPortNo <> 0)THEN

			eTCPState := E_TCPIP_DISCONNECT;
		END_IF


	(* close TCP connection *)
	E_TCPIP_DISCONNECT:

		(* TCP port has been closed *)
		IF eSocketState = eSOCKET_DISCONNECTED THEN

			eTCPState := E_TCPIP_IDLE;
		END_IF

(* unknown state *)
ELSE

	eTCPState := E_TCPIP_IDLE;
END_CASE


(* TCP port connection ctrl *)
fbTCPPortCtrl(
	sSrvNetID	:= '',
	nMode		:= LISTEN_MODE_CLOSEALL, (*LISTEN_MODE_USEOPENED, CONNECT_MODE_ENABLEDBG, LISTEN_MODE_CLOSEALL*)
	sRemoteHost	:= strTargetIPAddr,
	nRemotePort	:= nTargetPortNo,
	bEnable		:= eTCPState = E_TCPIP_CONNECT,
	tReconnect	:= tReconnectTime,
	bError		=> bError,
	nErrID		=> ,
	hSocket		=> hSocket,
	eState		=> eSocketState
);

IF NOT  fbTCPPortCtrl.bBusy THEN
	nErrorID := fbTCPPortCtrl.nErrId;
END_IF
(* connected status *)
bConnected := eSocketState = eSOCKET_CONNECTED;

END_FUNCTION_BLOCK

// ---- POUs/METS/Common LIB/09_SYSTEM LIB/FB_SYSTEM_AverageTimeDiff.TcPOU
FUNCTION_BLOCK FB_SYSTEM_AverageTimeDiff
VAR_INPUT
	bEnable : BOOL;
	bStart : BOOL;
	bStop :BOOL;
END_VAR
VAR_OUTPUT
	tLastDiff : TIME;
	tAverageDiff : TIME;
	arrTimeDiff : ARRAY[0..9] OF TIME;
END_VAR
VAR
	nIndex : INT;
	nCounter : INT;

	tTimeStop : TIME;
	tTimeStart : TIME;
	tTotalTime : TIME;

	fileTimeStart : T_FILETIME;
	fileTimeStop : T_FILETIME;

	fbStartTrig : R_TRIG;
	fbStopTrig : R_TRIG;
	fbCountTrig : R_TRIG;
	(*fbAvgTrig : R_TRIG;*)

	fbGetSystemTime : GETSYSTEMTIME;
END_VAR

IF bEnable THEN
	fbStartTrig(CLK := bStart);
	fbStopTrig(CLK := bStop);

	IF fbStartTrig.Q THEN
		fbGetSystemTime(timeLoDW => fileTimeStart.dwLowDateTime,
						timeHiDW => fileTimeStart.dwHighDateTime);
		tTimeStart := F_SYSTEM_StringToTime(fileTimeStart);
	END_IF;

	IF fbStopTrig.Q THEN
		fbGetSystemTime(timeLoDW => fileTimeStop.dwLowDateTime,
						timeHiDW => fileTimeStop.dwHighDateTime);
		tTimeStop := F_SYSTEM_StringToTime(fileTimeStop);
	END_IF;

	fbCountTrig(CLK := tTimeStop > tTimeStart AND NOT fbStartTrig.Q AND NOT fbStopTrig.Q);

	IF  fbCountTrig.Q THEN
		tLastDiff := tTimeStop - tTimeStart;
		MEMMOVE(ADR(arrTimeDiff[1] ), ADR(arrTimeDiff[0] ), SIZEOF(arrTimeDiff) -SIZEOF(arrTimeDiff[0] ) );
		arrTimeDiff[0] := tLastDiff;
		tTotalTime := tTotalTime + arrTimeDiff[0] ;
		nCounter := nCounter + 1;
	END_IF

	IF nCounter >=10 THEN
		tAverageDiff := tTotalTime / nCounter;
	END_IF
ELSE

	MEMSET(ADR(arrTimeDiff), 16#00, SIZEOF(arrTimeDiff));
	nCounter := 0;
	nIndex := 0;
	tTotalTime := T#0h0m0s0ms;
	tAverageDiff := T#0h0m0s0ms;
END_IF;

END_FUNCTION_BLOCK

// ---- POUs/METS/Common LIB/09_SYSTEM LIB/FB_SYSTEM_BarcodeType.TcPOU
(* decodes GS1-encoded barcode to determine if it is Code128 or DMC *)
FUNCTION_BLOCK FB_SYSTEM_BarcodeType
VAR_INPUT
	bExecute					: BOOL;		(* set TRUE to decode strGS1Barcode *)
	sCodeString				: STRING(255);	(* GS1-encoded string *)
	bRemoveFNC1				: BOOL;
	stCodeInfo_Pack			: ST_CodeInfo;
	stCodeInfo_Intermediate 	: ST_CodeInfo;
	stCodeInfo_Outer			: ST_CodeInfo;
	stCodeInfo_Case			: ST_CodeInfo;
	stPCMStatus				: ST_PCM_Status;
END_VAR
VAR_OUTPUT
	bDone					: BOOL;		(* TRUE = complete *)
	bPackBarcode				: BOOL;
	bOuterIntermediateBarcode	: BOOL;
	bOuterBarcode				: BOOL;
	bCaseBarcode				: BOOL;
	sPackBarcode				: T_PACK_Barcode;
	sOuterIntermediateBarcode	: STRING(255);
	sOuterBarcode				: T_OUTER_Barcode;
	sCaseBarcode				: T_CASE_Barcode;
END_VAR
VAR
	fbExecute			: R_TRIG;
	sNonGS1String	: STRING(255);
	nNonGS1Length	: INT;
	sGS1String		: STRING(255);	(* GS1-encoded string *)
	nGS1Length		: INT;
	eCodeAIType		: E_CodeAIType;
	fbDecodeGS1				: FB_SCANNER_DecodeGS1;
END_VAR

(* rising edge of bExecute *)
fbExecute(CLK := bExecute);

(* barcode read *)
IF fbExecute.Q = TRUE THEN

	(* clear outputs *)
	bDone := FALSE;
	bPackBarcode := FALSE;
	sPackBarcode := '';
	bOuterIntermediateBarcode	:= FALSE;
	sOuterIntermediateBarcode := '';
	bOuterBarcode := FALSE;
	sOuterBarcode := '';
	bCaseBarcode := FALSE;
	sCaseBarcode := '';

	sNonGS1String := SEL(bRemoveFNC1, sCodeString, F_ReplaceSingleChar(sCodeString, '$1D', ''));
	nNonGS1Length := LEN(sNonGS1String);

	fbDecodeGS1(strGS1String := CONCAT(']d2',sCodeString), bDontParseAsGS1 := FALSE, strBarcode => sGS1String);
	nGS1Length := LEN(sGS1String);

	IF stPCMStatus.sPackGTIN = F_CODE_GetItem(sGS1String, eCodeAIType.GTIN, stCodeInfo_Pack) AND stPCMStatus.sPackGTIN <> '' THEN
		sPackBarcode := SEL(fbDecodeGS1.strBarcode ='', sGS1String, sNonGS1String);
		bPackBarcode := TRUE;

	ELSIF stPCMStatus.sOuterGTIN = F_CODE_GetItem(sGS1String, eCodeAIType.GTIN, stCodeInfo_Outer) AND stPCMStatus.sOuterGTIN <> '' THEN
		sOuterBarcode := sGS1String;
		bOuterBarcode := TRUE;

	ELSIF stPCMStatus.sCaseGTIN = F_CODE_GetItem(sGS1String, eCodeAIType.GTIN, stCodeInfo_Case) AND stPCMStatus.sCaseGTIN <> '' THEN
		sCaseBarcode := sGS1String;
		bCaseBarcode := TRUE;

	ELSIF LEFT(stPCMStatus.sPackBrandSpec, stCodeInfo_Pack.stBrandSpecification.nCodeLength) = F_CODE_GetItem(sNonGS1String, eCodeAIType.BrandSpecification, stCodeInfo_Pack) AND
					stPCMStatus.sPackBrandSpec <> '' THEN
		sPackBarcode := sNonGS1String;
		bPackBarcode := TRUE;

	ELSIF LEFT(stPCMStatus.sOuterBrandSpec, stCodeInfo_Intermediate.stBrandSpecification.nCodeLength) = F_CODE_GetItem(sNonGS1String, eCodeAIType.BrandSpecification, stCodeInfo_Intermediate) AND
					stCodeInfo_Intermediate.stBrandSpecification.nListPosition <> 0 THEN
		sOuterIntermediateBarcode := sNonGS1String;
		bOuterIntermediateBarcode := TRUE;


	ELSIF LEFT(stPCMStatus.sOuterBrandSpec, stCodeInfo_Outer.stBrandSpecification.nCodeLength) = F_CODE_GetItem(sNonGS1String, eCodeAIType.BrandSpecification, stCodeInfo_Outer) AND
					stPCMStatus.sOuterBrandSpec <> '' THEN
		sOuterBarcode := sNonGS1String;
		bOuterBarcode := TRUE;

	ELSIF LEFT(stPCMStatus.sCaseBrandSpec, stCodeInfo_Case.stBrandSpecification.nCodeLength) = F_CODE_GetItem(sNonGS1String, eCodeAIType.BrandSpecification, stCodeInfo_Case) AND
					stPCMStatus.sCaseBrandSpec <> '' THEN
		sCaseBarcode := sNonGS1String;
		bCaseBarcode := TRUE;

	ELSIF nNonGS1Length = stCodeInfo_Pack.nEntireLength AND fbDecodeGS1.strBarcode ='' THEN
		sPackBarcode := sNonGS1String;
		bPackBarcode := TRUE;

	ELSIF nGS1Length = stCodeInfo_Pack.nEntireLength AND fbDecodeGS1.strBarcode <> '' THEN
		sPackBarcode := sGS1String;
		bPackBarcode := TRUE;

	ELSIF nNonGS1Length = stCodeInfo_Intermediate.nEntireLength  AND fbDecodeGS1.strBarcode ='' THEN
		sOuterIntermediateBarcode := sNonGS1String;
		bOuterIntermediateBarcode := TRUE;

	ELSIF nGS1Length = stCodeInfo_Intermediate.nEntireLength AND fbDecodeGS1.strBarcode <> '' THEN
		sOuterIntermediateBarcode := sGS1String;
		bOuterIntermediateBarcode := TRUE;

	ELSIF nNonGS1Length = stCodeInfo_Outer.nEntireLength  AND fbDecodeGS1.strBarcode ='' THEN
		sOuterBarcode := sNonGS1String;
		bOuterBarcode := TRUE;

	ELSIF nGS1Length = stCodeInfo_Outer.nEntireLength AND fbDecodeGS1.strBarcode <> '' THEN
		sOuterBarcode := sGS1String;
		bOuterBarcode := TRUE;

	ELSIF nNonGS1Length = stCodeInfo_Case.nEntireLength AND fbDecodeGS1.strBarcode ='' THEN
		sCaseBarcode := sNonGS1String;
		bCaseBarcode := TRUE;

	ELSIF nGS1Length = stCodeInfo_Case.nEntireLength  AND fbDecodeGS1.strBarcode <> '' THEN
		sCaseBarcode := sGS1String;
		bCaseBarcode := TRUE;
	END_IF

	IF stCodeInfo_Outer.stBrandSpecification.nListPosition <> 0  						AND
			stCodeInfo_Intermediate.stBrandSpecification.nListPosition = 0 				AND
			stCodeInfo_Outer.nEntireLength = stCodeInfo_Intermediate.nEntireLength 	THEN

		sOuterIntermediateBarcode := sOuterBarcode;
		bOuterIntermediateBarcode := bOuterBarcode;
	END_IF


	(* update output *)
	bDone := TRUE;

(* bExecute has been reset *)
ELSIF bExecute = FALSE THEN

	(* reset output *)
	bDone := FALSE;
END_IF

END_FUNCTION_BLOCK

// ---- POUs/METS/Common LIB/09_SYSTEM LIB/FB_SYSTEM_DateTime.TcPOU
(* generates PLC and System time clocks in real-time kernel, synchronise to System time when required *)
FUNCTION_BLOCK FB_SYSTEM_DateTime
VAR_INPUT
	bEnable					: BOOL;		(* set TRUE to enable system time update *)
	bNVDataInitOK			: BOOL;		(* set TRUE when NV data is initialised, enables PCM timer *)
	nShiftOffsetTime		: DINT;		(* OffsetTime = SystemTime + tTimeOffset*)
END_VAR
VAR_IN_OUT
	stPCMStatus				: ST_PCM_Status;	(* PCM status *)
	(*stMetsStatusNV			: ST_NOVRAM_CaseTraceNV;	(* CaseTrace NV data, used for last PCM  timestamps *)*)
END_VAR
VAR_OUTPUT
	bSystemTimeValid		: BOOL;		(* TRUE = System time is valid *)
	bPCMTimeValid			: BOOL;		(* TRUE = PCM time is valid *)
	bBusy					: BOOL;		(* TRUE = sync in progress, PLC continues to be updated while sync is active *)
	stCTDateTime				: ST_SYSTEM_DateTime;	(* output time structure *)
END_VAR
VAR
	fbSyncSysTime			: FB_SquareWave;
	fbInitPCMTime			: R_TRIG;
	fbSyncPCMTime			: R_TRIG;
	bSyncPCMTime			: BOOL;

	eState					: E_SYSTEM_CTState;
	eErrorState				: E_SYSTEM_CTState;
	fbReadSystemTime		: NT_GetTime;
	fbGetTimeZoneInfo		: FB_GetTimeZoneInformation;
	eTimeZoneID				: E_TimeZoneID;
	sTimeZoneInfo			: ST_TimeZoneInformation;
	sBaseTime				: TIMESTRUCT;

	bStartSystemTimer		: BOOL;
	fbSystemTime			: RTC_EX2;
	nLastSysSecond			: WORD;
	nSysUpdateStep			: UINT;
	nSystemTime				: T_Filetime;
	nLastTime				: T_Filetime;

	bStartPCMTimer			: BOOL;
	fbPCMTime				: RTC_EX2;
	bSyncPCMToSysTime		: BOOL;

END_VAR
(*
-------------------------------------------------------------------------------------------------
Date		Version	Author	Comments
-------------------------------------------------------------------------------------------------
01/08/2014	2.00.00	PB		sPLCTime added as VAR_IN_OUT to allow last value to be stored in NOVRAM.
							At start-up, sPLCTime is now initialised to stored sPLCTime or sSystemTime, whichever is later.
							sPLCTime is only synchronised with sSystemDate time on rising edge of bUpdatePLCTime.
							These changes prevent sPLCTime from jumping back in time and remove the possibility of producing duplicate timestamp codes.
							sUTCTime and corresponding date and time strings added.
							nUTCOffset also generated to determine the time difference between sSystemTime and sUTCTime, specified in ms.

-------------------------------------------------------------------------------------------------
03/08/2012	1.39.00	PB		Re-written to generate PLC, System and Offset time and create updated ST_SYSTEM_DateTime structure.
							PLC time is synchronised at start-up and on rising edge of bSyncPLCTime.
							System time is synchronised at start-up and every 1s thereafter.
							Offset time is System time with tTimeOffset subtracted.
16/12/2011	1.36.00	PB		Initial release

-------------------------------------------------------------------------------------------------
*)

(* enabled *)
IF bEnable = TRUE THEN

	(* re-sync sSystemTime system every 1s *)
	fbSyncSysTime(
		bEnable		:= bStartSystemTimer,
		tPeriod		:= T#1s,
	);

	(* synchronise sPCMTime when PCM is enabled OR RetailSKU is changed *)
	fbInitPCMTime(CLK := bNVDataInitOK AND stPCMStatus.bEnabled);
	fbSyncPCMTime(CLK := bNVDataInitOK AND stPCMStatus.bRSKUChanged);

	(* PCM enabled *)
	IF fbInitPCMTime.Q = TRUE THEN

		(* PCM time will be synchronised to SystemTime or LastPCMTime used, whichever is later *)
		bSyncPCMTime := TRUE;
		(* this ensures that PCM time continues from last time-stamp used to prevent duplicate timestamp codes *)

	(* PCM RetailSKU has changed *)
	ELSIF fbSyncPCMTime.Q = TRUE THEN

		(* clear last PCM time *)
		MEMSET(ADR(stPCMStatus.stLastPCMTime), 16#00, SIZEOF(stPCMStatus.stLastPCMTime));

		(* PCM time will be synchronised to SystemTime as LastPCMTime will be older than SystemTime*)
		bSyncPCMTime := TRUE;
		(* bRSKUChanged is suppressed when PCM is first loaded *)
	END_IF

	CASE eState OF

		(* INIT state *)
		E_SYSTEMCT_IDLE:

			(* system timer not initialised *)
			IF stCTDateTime.bSystemTimeValid = FALSE THEN

				(* update output and clear error state *)
				bBusy := TRUE;
				eErrorState := eState;

				eState := E_SYSTEMCT_TIMEZONE;

			(* system timer initialised *)
			ELSE

				(* re-sync system timer *)
				IF fbSyncSysTime.bRisingEdge = TRUE OR bSyncPCMTime = TRUE THEN

					(* update output and clear error state *)
					bBusy := TRUE;
					eErrorState := eState;

					eState := E_SYSTEMCT_TIMEZONE;
				END_IF
			END_IF


		(* get timezone info *)
		E_SYSTEMCT_TIMEZONE:
			(* read time zone info from conifg file*)
			(*stCTDateTime.nSystemTimeOffset := nShiftOffsetTime;

			eState := E_SYSTEMCT_SYSTEMTIME;*)

			(* read Windows time zone info *)
			fbGetTimeZoneInfo(
				sNetID		:= '',
				bExecute	:= TRUE,
				tTimeout	:= T#5s
			);

			(* read timezone complete *)
			IF fbGetTimeZoneInfo.bBusy = FALSE THEN

				(* read timezone completed OK *)
				IF fbGetTimeZoneInfo.bError = FALSE THEN

					(* get time zone info *)
					eTimeZoneID := fbGetTimeZoneInfo.tzID;
					sTimeZoneInfo := fbGetTimeZoneInfo.tzInfo;

					(* Daylight Saving time active *)
					IF eTimeZoneID = eTimeZoneID_Daylight THEN

						(* convert mins to ms *)
						stCTDateTime.nSystemTimeOffset := (sTimeZoneInfo.bias + sTimeZoneInfo.daylightBias) * -60000;

					(* Standard time active *)
					ELSIF eTimeZoneID = eTimeZoneID_Standard THEN

						(* convert mins to ms *)
						stCTDateTime.nSystemTimeOffset := (sTimeZoneInfo.bias + sTimeZoneInfo.standardBias) * -60000;

					(* eTimeZoneID invalid *)
					ELSE

						(*stCTDateTime.nSystemTimeOffset := 0;*)
						stCTDateTime.nSystemTimeOffset := nShiftOffsetTime;
					END_IF

					stCTDateTime.sUTCTimeZoneOffset  := F_SYSTEM_SystemTimeOffsetToHHMM(stCTDateTime.nSystemTimeOffset);


					eState := E_SYSTEMCT_SYSTEMTIME;

				(* read timezone error *)
				ELSE

					eErrorState := eState;

					eState := E_SYSTEMCT_ERROR;
				END_IF

				(* close off fbGetTimeZoneInfo *)
				fbGetTimeZoneInfo(bExecute := FALSE);
			END_IF


		E_SYSTEMCT_SYSTEMTIME:

			(* read system time *)
			fbReadSystemTime(
				NETID	:= '',
				START	:= TRUE,
				TMOUT	:= T#1s
			);

			(* read system time complete and sPLCTime has been restored *)
			IF fbReadSystemTime.BUSY = FALSE THEN

				(* read system time completed OK *)
				IF fbReadSystemTime.ERR = FALSE THEN

					(* base time for updating system time *)
					sBaseTime := fbReadSystemTime.TIMESTR;
					bStartSystemTimer := TRUE;

					(* re-sync system time *)
					fbSystemTime(EN := FALSE);
	
					(* re-sync PCM time *)
					IF bSyncPCMTime = TRUE THEN

						bSyncPCMTime := FALSE;
						bStartPCMTimer := TRUE;

						(* convert sLastPCMTimeStamp and current system time from TIMESTRUCT to T_Filetime *)
						nLastTime := SYSTEMTIME_TO_FILETIME(stPCMStatus.stLastPCMTime);
						nSystemTime := SYSTEMTIME_TO_FILETIME(fbReadSystemTime.TIMESTR);
	
						(* sLastPCMTimeStamp > sSystemTime *)
						IF nLastTime.dwHighDateTime > nSystemTime.dwHighDateTime OR (nLastTime.dwHighDateTime = nSystemTime.dwHighDateTime AND nLastTime.dwLowDateTime > nSystemTime.dwLowDateTime) THEN
	
							(* sync PCM time to last PCM time stamp + 1s *)
							bSyncPCMToSysTime := FALSE;
	
						(* sLastPCMTimeStamp <= sSystemTime *)
						ELSE
	
							(* sync PCM time to system time *)
							bSyncPCMToSysTime := TRUE;
						END_IF
	
						(* re-sync PCM PLC time *)
						fbPCMTime(EN := FALSE);
					END_IF

					eState := E_SYSTEMCT_DONE;

				(* read system time error *)
				ELSE
	
					eErrorState := eState;
	
					eState := E_SYSTEMCT_ERROR;
				END_IF

				(* close off fbReadSystemTime *)
				fbReadSystemTime(START := FALSE);
			END_IF
	
	
		(* done *)
		E_SYSTEMCT_DONE:
	
			(* update outputs *)
			bBusy := FALSE;
	
			eState := E_SYSTEMCT_IDLE;
	

	(* unknown state *)
	ELSE
	
		eState := E_SYSTEMCT_IDLE;
	END_CASE
	
	
	(* system timer - sync occurs when EN goes TRUE *)
	fbSystemTime(
		EN		:= bEnable AND bStartSystemTimer,
		PDT		:= sBaseTime,
		PMICRO	:= 0,
		Q		=> stCTDateTime.bSystemTimeValid,
		CDT		=> stCTDateTime.sSystemTime
	);

	(* system timer not active *)
	IF fbSystemTime.EN = FALSE OR stCTDateTime.bSystemTimeValid = FALSE THEN

		(* clear sSystemTime, sOffsetTime and sUTCTime *)
		stCTDateTime.bSystemTimeValid := FALSE;
		MEMSET(ADR(stCTDateTime.sSystemTime), 16#00, SIZEOF(stCTDateTime.sSystemTime));
		MEMSET(ADR(stCTDateTime.sOffsetTime), 16#00, SIZEOF(stCTDateTime.sOffsetTime));
		MEMSET(ADR(stCTDateTime.sUTCTime), 16#00, SIZEOF(stCTDateTime.sUTCTime));

	(* system date/time is valid *)
	ELSE
	
		(* system update step *)
		CASE nSysUpdateStep OF
	
			(* idle *)
			0:
	
				(* system time second has changed *)
				IF stCTDateTime.sSystemTime.wSecond <> nLastSysSecond THEN
	
					(* move next step and remember current second *)
					nSysUpdateStep := nSysUpdateStep + 1;
					nLastSysSecond := stCTDateTime.sSystemTime.wSecond;
				END_IF
	
			(* update sOffsetTime *)
			1:

				(* apply offset to sSystemTime to produce sOffsetTime *)
				stCTDateTime.sOffsetTime := F_ApplyTimeOffset(stCTDateTime.sSystemTime, nShiftOffsetTime);
				stCTDateTime.sOffsetTime.wMilliseconds := 0;
				nSysUpdateStep := nSysUpdateStep + 1;

	
			(* update sUTCTime *)
			2:

				(* apply offset to sSystemTime to produce UTC time *)
				stCTDateTime.sUTCTime := F_ApplyTimeOffset(stCTDateTime.sSystemTime, stCTDateTime.nSystemTimeOffset *-1);
				stCTDateTime.sUTCTime.wMilliseconds := 0;
				(*stCTDateTime.sUTCTimeZoneOffset := strUTCTimeZone;*)
				nSysUpdateStep := nSysUpdateStep + 1;

			(* generate HMI date/time display string *)
			3:
	
				stCTDateTime.strHMIDateTime := F_SYSTEM_HMIDateTime(stCTDateTime.sSystemTime);
				nSysUpdateStep := nSysUpdateStep + 1;
	
		(* unkonw state *)
		ELSE
	
			(* return to step 0 *)
			nSysUpdateStep := 0;
		END_CASE
	END_IF


	(* PCM timer - sync occurs bStartPCMTimer is set to TRUE *)
	fbPCMTime(
		EN		:= stPCMStatus.bEnabled AND bStartPCMTimer,
		PDT		:= SEL(bSyncPCMToSysTime, stPCMStatus.stLastPCMTime, stCTDateTime.sSystemTime),
		PMICRO	:= 0,
		Q		=> stCTDateTime.bPCMTimeValid,
		CDT		=> stCTDateTime.sPCMTime
	);

	(* PCM timer not active *)
	IF fbPCMTime.EN = FALSE OR bPCMTimeValid = FALSE THEN

		(* clear sPCMTime *)
		MEMSET(ADR(stCTDateTime.sPCMTime), 16#00, SIZEOF(stCTDateTime.sPCMTime));

	(* PCM timer active *)
	ELSE

		(* reduce timer resolution to 0.1s *)
		stCTDateTime.sPCMTime.wMilliseconds := (stCTDateTime.sPCMTime.wMilliseconds / 100) * 100;
	END_IF

(* disabled *)
ELSE

	(* clear outputs *)
	bBusy := FALSE;
	MEMSET(ADR(stCTDateTime), 16#00, SIZEOF(stCTDateTime));

	(* disable timers *)
	bStartSystemTimer := FALSE;
	bStartPCMTimer := FALSE;

END_IF

(* update outputs *)
(*stCTDateTime.sUTCTimeZoneOffset := strUTCTimeZone;*)

bSystemTimeValid := stCTDateTime.bSystemTimeValid;
bPCMTimeValid := stCTDateTime.bPCMTimeValid;

END_FUNCTION_BLOCK

// ---- POUs/METS/Common LIB/09_SYSTEM LIB/FB_SYSTEM_HardwareOS.TcPOU
(* returns CX Hardware type, Operating System and Hardware info *)
FUNCTION_BLOCK FB_SYSTEM_HardwareOS
VAR_INPUT
	bExecute			: BOOL;		(* set TRUE to read CX hardware and OS info *)
	sBaseFolder		: STRING(31);	(* base folder for system (without disk ref) *)
END_VAR
VAR_OUTPUT
	bDone			: BOOL;		(* TRUE = complete *)
	bBusy			: BOOL;		(* TRUE = in progress *)
	bError			: BOOL;		(* TRUE = error *)
	nErrorID			: UDINT;	(* error ID *)
	bBasePathOK		: BOOL;		(* base path checked OK *)
	sBasePath		: T_FolderPath;	(* base folder with disk ref added *)
	sTCInstalationPath : T_FolderPath;
	eHWType			: E_CX_HWType;	(* hardware type *)
	eOSType			: E_SYSTEM_OSType;		(* OS type *)
	stHardware		: ST_CxDeviceIdentificationEx;	(* hardware info *)
END_VAR
VAR
	fbExecute			: R_TRIG;
	eState			: E_CX_State;
	eErrorState		: E_CX_State;

	fbHardware		: FB_CxGetDeviceIdentificationEx;
	fbReadRegKey		: FB_RegQueryValue;

	fbFindFolder		: FB_EnumFindFileEntry;
	eCmdType		: E_EnumCmdType;
END_VAR

(* monitor bExecute *)
fbExecute(CLK := bExecute);

CASE eState OF

	(* idle *)
	E_CX_State.IDLE:

		(* rising edge of bExecute *)
		IF fbExecute.Q = TRUE THEN

			(* update outputs *)
			bDone := FALSE;
			bBusy := TRUE;
			bError := FALSE;
			nErrorID := 0;

			(* initalise vars *)
			bBasePathOK := FALSE;
			eCmdType := eEnumCmd_First;
			eErrorState := eState;

			eState := E_CX_State.HW;

		(* no action required *)
		ELSIF bExecute = FALSE THEN

			(* update outputs *)
			bDone := FALSE;
			bBusy := FALSE;
			bError := FALSE;
			nErrorID := 0;
		END_IF


	(* get hardware platform *)
	E_CX_State.HW:

		(* get hardware info *)
		fbHardware(
			bExecute	:= TRUE,
			tTimeout	:= T#1s
		);

		(* read hardware complete *)
		IF fbHardware.bBusy = FALSE THEN

			(* read hardware completed OK *)
			IF fbHardware.bError = FALSE THEN

				(* log hardware info *)
				stHardware := fbHardware.stDevIdent;

				(* platform is CX1 *)
				IF LEFT(stHardware.strImageDevice, LEN('CX1')) = 'CX1' THEN

					eHWType := E_CX_HWType.CX1;

				(* platform is CX2 *)
				ELSIF LEFT(stHardware.strImageDevice, LEN('CX2')) = 'CX2' THEN

					eHWType := E_CX_HWType.CX2;

				(* platform is CX5 *)
				ELSIF LEFT(stHardware.strImageDevice, LEN('CX5')) = 'CX5' THEN

					eHWType := E_CX_HWType.CX5;

				(* platform is CX8 *)
				ELSIF LEFT(stHardware.strImageDevice, LEN('CX8')) = 'CX8' THEN

					eHWType := E_CX_HWType.CX8;

				(* platform is CX9 *)
				ELSIF LEFT(stHardware.strImageDevice, LEN('CX9')) = 'CX9' THEN

					eHWType := E_CX_HWType.CX9;
					
				(* platform is CP *)
				ELSIF LEFT(stHardware.strImageDevice, LEN('CB')) = 'CB' THEN

					eHWType := E_CX_HWType.CP;
					
				(* platform assumed to be PC *)
				ELSE

					eHWType := E_CX_HWType.PC;
				END_IF
			END_IF

			eState := E_CX_State.OS;

			fbHardware(bExecute	:= FALSE);
		END_IF


	(* check operating system *)
	E_CX_State.OS:

		(* read registry key *)
		fbReadRegKey(
			sNetId		:= '',
			sSubKey		:= 'SYSTEM\CurrentControlSet\Control\Session Manager\Environment',
			sValName	:= 'TWINCAT3DIR',
			cbData		:= SIZEOF(sTCInstalationPath),
			pData		:= ADR(sTCInstalationPath),
			bExecute	:= TRUE,
			tTimeOut	:= T#1s
		);

		(* read registry key complete *)
		IF fbReadRegKey.bBusy = FALSE THEN

			(* read registry key completed OK *)
			IF fbReadRegKey.bError = FALSE THEN

				(* value on WinCE will be '\Hard Disk\TwinCAT' *)
				IF sTCInstalationPath = '\Hard Disk\TwinCAT' THEN

					(* OS is WinCE *)
					eOSType := E_OS_WINCE;
					sBasePath := CONCAT('\Hard Disk\', sBaseFolder);

				(* other value *)
				ELSE

					(* OS is full Windows *)
					eOSType := E_OS_WINDOWS;
					sBasePath := CONCAT('C:\', sBaseFolder);
				END_IF

				(* strBaseFolder is terminated with '\' char *)
				IF RIGHT(sBasePath, 1) = '\' THEN

					(* remove '\' from end of strBasePath for folder check *)
					sBasePath := LEFT(sBasePath, LEN(sBasePath) - 1);
				END_IF

				eState := E_CX_State.BASEFOLDER;

			(* read registry key error *)
			ELSE

				(* update outputs *)
				bError := TRUE;
				nErrorID := fbReadRegKey.nErrId;
				eErrorState := eState;

				eState := E_CX_State.DONE;
			END_IF

			(* close off fbReadRegKey *)
			fbReadRegKey(bExecute := FALSE);
		END_IF


	(* check base folder *)
	E_CX_State.BASEFOLDER:

		(* find folder *)
		fbFindFolder(
			sNetId		:= '',
			sPathName	:= sBasePath,
			eCmd		:= eCmdType,
			bExecute	:= TRUE,
			tTimeout	:= T#1s
		);

		(* find folder complete *)
		IF fbFindFolder.bBusy = FALSE THEN

			(* find folder completed OK *)
			IF fbFindFolder.bError = FALSE THEN

				(* folder found *)
				IF fbFindFolder.stFindFile.fileAttributes.bDirectory = TRUE THEN

					(* base path OK, cancel fbFindFolder *)
					bBasePathOK := TRUE;
					eCmdType := eEnumCmd_Abort;

					(* last char of strBasePath is not '\' *)
					IF RIGHT(sBasePath, 1) <> '\' THEN

						(* re-apply '\' char to end of strBasePath *)
						sBasePath := CONCAT(sBasePath, '\');
					END_IF

				(* end of list *)
				ELSIF fbFindFolder.bEOE = TRUE THEN

					(* Windows platform and base folder not found on C: drive *)
					IF eOSType = E_OS_WINDOWS AND LEFT(sBaseFolder, 3) = 'C:\' THEN

						(* check for base folder on D drive *)
						sBasePath := CONCAT('D:\', sBaseFolder);

					(* end of search *)
					ELSE

						(* base path not found *)
						IF bBasePathOK = FALSE THEN

							(* clear path and update output *)
							sBasePath := '';
							bError := TRUE;
						END_IF

						eState := E_CX_State.DONE;
					END_IF
				END_IF

			(* find folder completed OK *)
			ELSE

				(* update outputs *)
				bError := TRUE;
				nErrorID := fbFindFolder.nErrID;
				eErrorState := eState;

				eState := E_CX_State.DONE;
			END_IF

			(* close off fbFindFolder *)
			fbFindFolder(bExecute := FALSE);
		END_IF


	(* done *)
	E_CX_State.DONE:

		(* update outputs *)
		bBusy := FALSE;
		bDone := TRUE;

		eState := E_CX_State.IDLE;

(* unknown state *)
ELSE

	eState := E_CX_State.IDLE;
END_CASE

END_FUNCTION_BLOCK

// ---- POUs/METS/Common LIB/09_SYSTEM LIB/FB_SYSTEM_MachineState.TcPOU
FUNCTION_BLOCK FB_SYSTEM_MachineState
VAR_INPUT
	bPowerUpComplete				:BOOL;
	bNoActiveAlarms				:BOOL;
	bSafetyRelayOK				: BOOL;
	bMachnieManual				: BOOL;
	bMachineReadyToStart				: BOOL;
	bStartRequest					: BOOL;
	bMachineRunning				: BOOL;
	bMachineConditionalRunning		: BOOL;
	bConveorMode				: BOOL;
	bStopRequest					: BOOL;
	bMachineStopped				: BOOL;
	bForceMachineState				: BOOL := FALSE;
	nForcedMachineState			: INT;
END_VAR
VAR_OUTPUT
	eMachineState					: E_SYSTEM_MachineState;
	stMachineState					: ST_SYSTEM_MachineState;
	sMachineState					: STRING;
	bMachineStateChanged		: BOOL;
	bStoppingTimeOut				: BOOL;
END_VAR
VAR
	tonSystemInitialisingDebounce	: TON;
	tonSystemInitialisingTimeout		: TON;
	tonSystemStoppingTimeout		: TON;
	sLastMachineState					: STRING;
END_VAR
VAR CONSTANT
	(* list of supported machine states *)
	aMachineState			: ARRAY[1..12] OF STRING :=[
												'POWERUP',
												'IMMEDIATE STOPPED',
												'MACHINE IN ERROR',
												'INITIALISING',
												'MANUAL',
												'READY TO START',
												'STOPPING',
												'RUNNING',
												'WAITING FOR PRODUCT',
												'PASSTHROUGH ACTIVE',
												'CONDITIONAL RUNNING'];
END_VAR

(********************************(Force Machine State)**********************************************************)
IF bForceMachineState THEN

	CASE	nForcedMachineState OF
	0:
		eMachineState					:= E_SYSTEM_MachineState.POWERUP;
	100:
		eMachineState					:=E_SYSTEM_MachineState.IMMEDIATESTOPPED;
	110:
		eMachineState					:=E_SYSTEM_MachineState.MACHINEINERROR;
	200:
		eMachineState					:=E_SYSTEM_MachineState.INITIALISING;
	210:
		eMachineState					:=E_SYSTEM_MachineState.MANUAL;
	300:
		eMachineState					:=E_SYSTEM_MachineState.READYTOSTART;
	310:
		eMachineState					:=E_SYSTEM_MachineState.STOPPING;
	400:
		eMachineState					:=E_SYSTEM_MachineState.RUNNING;
	410:
		eMachineState					:=E_SYSTEM_MachineState.WAITINGFORPRODUCT;
	420:
		eMachineState					:=E_SYSTEM_MachineState.PASSTHROUGHACTIVE;
	430:
		eMachineState					:=E_SYSTEM_MachineState.CONDITIONALRUNNING;
	ELSE
		eMachineState					:=E_SYSTEM_MachineState.POWERUP;
	END_CASE

stMachineState.bSystemPowerUp 						:=	(eMachineState=E_SYSTEM_MachineState.POWERUP);
IF stMachineState.bSystemPowerUp THEN 			sMachineState := aMachineState[1]; END_IF

stMachineState.bImmediateStopped 					:=	(eMachineState=E_SYSTEM_MachineState.IMMEDIATESTOPPED);
IF stMachineState.bImmediateStopped THEN 			sMachineState := aMachineState[2]; END_IF

stMachineState.bMachineInError 						:=	(eMachineState=E_SYSTEM_MachineState.MACHINEINERROR);
IF stMachineState.bMachineInError THEN 			sMachineState := aMachineState[3]; END_IF

stMachineState.bSystemInitialising 					:=	(eMachineState=E_SYSTEM_MachineState.INITIALISING);
IF stMachineState.bSystemInitialising THEN 			sMachineState := aMachineState[4]; END_IF

stMachineState.bManualMode 							:=	(eMachineState=E_SYSTEM_MachineState.MANUAL);
IF stMachineState.bManualMode THEN 			sMachineState := aMachineState[5]; END_IF

stMachineState.bSystemReadyToStart 					:=	(eMachineState=E_SYSTEM_MachineState.READYTOSTART);
IF stMachineState.bSystemReadyToStart THEN 			sMachineState := aMachineState[6]; END_IF

stMachineState.bSystemCycleStopping				:=	(eMachineState=E_SYSTEM_MachineState.STOPPING);
IF stMachineState.bSystemCycleStopping THEN 			sMachineState := aMachineState[7]; END_IF

stMachineState.bSystemRunning						:=	(eMachineState=E_SYSTEM_MachineState.RUNNING);
IF stMachineState.bSystemRunning THEN 			sMachineState := aMachineState[8]; END_IF

stMachineState.bMachineWaitingForProduct 			:=	(eMachineState=E_SYSTEM_MachineState.WAITINGFORPRODUCT);
IF stMachineState.bMachineWaitingForProduct THEN 			sMachineState := aMachineState[9]; END_IF

stMachineState.bMachineInConditionalRun 			:=	(eMachineState=E_SYSTEM_MachineState.CONDITIONALRUNNING);
IF stMachineState.bMachineInConditionalRun THEN 			sMachineState := aMachineState[10]; END_IF

stMachineState.bTrackAndTraceDeactivated			:=	(eMachineState=E_SYSTEM_MachineState.PASSTHROUGHACTIVE);
IF stMachineState.bTrackAndTraceDeactivated THEN 			sMachineState := aMachineState[11]; END_IF


IF sLastMachineState <> sMachineState THEN

	bMachineStateChanged	:= TRUE;
	sLastMachineState := sMachineState;
ELSE
	bMachineStateChanged	:= FALSE;
END_IF;



RETURN;
END_IF

(********************************(Timers )**********************************************************)

(* System Initialising Timer *)
tonSystemInitialisingDebounce(
	IN:=(eMachineState=E_SYSTEM_MachineState.INITIALISING),
	PT:=T#1S,
	Q=>,
	ET=>
);

(* System Initialising Timeout Timer *)
(*tonSystemInitialisingTimeout(
	IN:=(eMachineState=E_SYSTEM_MachineState.INITIALISING),
	PT:=T#2M,
	Q=>,
	ET=>
);*)


(* System Stopping Timeout Timer *)
tonSystemStoppingTimeout(
	IN:=(eMachineState=E_SYSTEM_MachineState.STOPPING),
	PT:=T#2M,
	Q=>bStoppingTimeOut,
	ET=>
);

(********************************(Sequence )*******************************************************)
CASE	eMachineState OF

E_SYSTEM_MachineState.POWERUP:
	(* Move to Immediate Stopped once Power Up Timer has completed *)
	IF 		bPowerUpComplete		THEN
		eMachineState									:=	E_SYSTEM_MachineState.IMMEDIATESTOPPED;
	END_IF

E_SYSTEM_MachineState.IMMEDIATESTOPPED:
	(* Move to Immediate Fault once there is an Immediate Fault *)
	IF	 NOT	bNoActiveAlarms		THEN
		eMachineState									:=	E_SYSTEM_MachineState.MACHINEINERROR;
	(* Move to System Initialising once there is no Immediate Fault *)
	ELSIF		bNoActiveAlarms		THEN
		(*eMachineState									:=	E_SYSTEM_MachineState.STOPPING;*)
		eMachineState								:=	E_SYSTEM_MachineState.INITIALISING;
	END_IF

E_SYSTEM_MachineState.MACHINEINERROR:
	(* Move to System ImmedietStope  once there is no Immediate Fault *)
	IF		bNoActiveAlarms		THEN
		eMachineState									:=	E_SYSTEM_MachineState.IMMEDIATESTOPPED;
	END_IF

E_SYSTEM_MachineState.INITIALISING:
	(* Move to Immediate Stopped once there is an Immediate Fault  *) (* tonSystemInitialisingTimeout - trzeba dodac to do alarmow z timerem 0*)
	(*IF	(NOT 	bNoActiveAlarms 	AND tonSystemInitialisingDebounce.Q) OR tonSystemInitialisingTimeout.Q	THEN*)
	IF	NOT 	bNoActiveAlarms 	AND tonSystemInitialisingDebounce.Q	THEN
		eMachineState									:=	E_SYSTEM_MachineState.IMMEDIATESTOPPED;
	(* Move to Manual mode *)
	ELSIF		bNoActiveAlarms	AND 	bMachnieManual	THEN
		eMachineState									:=	E_SYSTEM_MachineState.MANUAL;
	(* Move to System Ready To Start once all Stations are Homed and the System Initialising Timer is Complete *)
	ELSIF		bNoActiveAlarms	AND 	bMachineReadyToStart	THEN
		eMachineState									:=	E_SYSTEM_MachineState.READYTOSTART;
	END_IF

E_SYSTEM_MachineState.MANUAL:
	(* Move to Immediate Stopped once there is an Immediate Fault  *) (* tonSystemInitialisingTimeout - trzeba dodac to do alarmow z timerem 0*)
	IF	(NOT bNoActiveAlarms	AND NOT bMachnieManual) OR NOT bSafetyRelayOK THEN
		eMachineState									:=	E_SYSTEM_MachineState.IMMEDIATESTOPPED;
	(* Move to System Initialising once there is no Immediate Fault and Manual mode disable*)
	ELSIF		bNoActiveAlarms 	AND NOT bMachnieManual	THEN
		eMachineState									:=	E_SYSTEM_MachineState.INITIALISING;
	END_IF

E_SYSTEM_MachineState.READYTOSTART:
	(* Move to Immediate Stopped once there is an Immediate Fault *)
	IF	NOT 	bNoActiveAlarms	THEN
		eMachineState									:=	E_SYSTEM_MachineState.IMMEDIATESTOPPED;
	ELSIF NOT bMachineReadyToStart	THEN
		eMachineState									:=	E_SYSTEM_MachineState.INITIALISING;
		(* Move to Manual mode *)
	ELSIF		bNoActiveAlarms	AND 	bMachnieManual	THEN
		eMachineState									:=	E_SYSTEM_MachineState.MANUAL;
	(* Move to System Auto if the Start Button has been pressed *)
	ELSIF		bStartRequest		(*AND	bMachineReadyToStart*)	THEN
		eMachineState									:=	E_SYSTEM_MachineState.RUNNING;
	END_IF

E_SYSTEM_MachineState.RUNNING:

	IF	bMachineConditionalRunning	AND NOT bStopRequest 	THEN
		eMachineState								:=	E_SYSTEM_MachineState.CONDITIONALRUNNING;
	(* Move to Immediate Stopped once there is an Immediate Fault *)
	ELSIF NOT bNoActiveAlarms			THEN
		eMachineState								:=	E_SYSTEM_MachineState.IMMEDIATESTOPPED;
	ELSIF bStopRequest					THEN
		eMachineState								:=	E_SYSTEM_MachineState.STOPPING;
	(* Move to Macine conveor mode only *)
	ELSIF bConveorMode				THEN
		eMachineState								:=	E_SYSTEM_MachineState.PASSTHROUGHACTIVE;
	(* Move to Macine waiting for producte once if is not running *)
	ELSIF	NOT bMachineRunning			THEN
		eMachineState								:=	E_SYSTEM_MachineState.WAITINGFORPRODUCT;
	END_IF

E_SYSTEM_MachineState.CONDITIONALRUNNING:
	(* Move to Immediate Stopped once there is an Immediate Fault   or  manual selector is in manual mode*)
	IF NOT bNoActiveAlarms AND NOT bMachineConditionalRunning	THEN
		eMachineState								:=	E_SYSTEM_MachineState.IMMEDIATESTOPPED;
	ELSIF		bStopRequest				THEN
		eMachineState								:=	E_SYSTEM_MachineState.STOPPING;
	(* Move to Macine conveor mode only *)
	ELSIF bConveorMode				THEN
		eMachineState								:=	E_SYSTEM_MachineState.PASSTHROUGHACTIVE;
	(* Move to System runnung state once machine is running*)
	ELSIF bMachineRunning				THEN
		eMachineState								:=	E_SYSTEM_MachineState.RUNNING;
	(* Move to Macine waiting for producte once if is not running *)
	ELSIF	NOT bMachineRunning AND NOT bMachineConditionalRunning	THEN
		eMachineState								:=	E_SYSTEM_MachineState.WAITINGFORPRODUCT;
	END_IF

E_SYSTEM_MachineState.WAITINGFORPRODUCT:
	IF	bMachineConditionalRunning	AND NOT bStopRequest 	THEN
		eMachineState								:=	E_SYSTEM_MachineState.CONDITIONALRUNNING;
	(* Move to Immediate Stopped once there is an Immediate Fault *)
	ELSIF NOT bNoActiveAlarms			THEN
		eMachineState								:=	E_SYSTEM_MachineState.IMMEDIATESTOPPED;
	ELSIF		bStopRequest				THEN
		eMachineState								:=	E_SYSTEM_MachineState.STOPPING;
	(* Move to Macine conveor mode only *)
	ELSIF bConveorMode				THEN
		eMachineState								:=	E_SYSTEM_MachineState.PASSTHROUGHACTIVE;
	(* Move to System runnung state once machine is running*)
	ELSIF bMachineRunning				THEN
		eMachineState								:=	E_SYSTEM_MachineState.RUNNING;
	END_IF

E_SYSTEM_MachineState.PASSTHROUGHACTIVE:
	(* Move to Immediate Stopped once there is an Immediate Fault   or  manual selector is in manual mode*)
	IF	NOT 	bNoActiveAlarms			THEN
		eMachineState								:=	E_SYSTEM_MachineState.IMMEDIATESTOPPED;
	ELSIF	 bStopRequest	(*OR NOT bConveorMode*)		THEN
		eMachineState								:=	E_SYSTEM_MachineState.STOPPING;
	ELSIF NOT bConveorMode				THEN
		eMachineState								:=	E_SYSTEM_MachineState.INITIALISING;
	END_IF

E_SYSTEM_MachineState.STOPPING:
	(* Move to Immediate Stopped once there is an Immediate Fault   or  manual selector is in manual mode*)
	IF	NOT 	bNoActiveAlarms			THEN
		eMachineState								:=	E_SYSTEM_MachineState.IMMEDIATESTOPPED;
	ELSIF		bMachineStopped			THEN
		eMachineState								:=	E_SYSTEM_MachineState.INITIALISING;
	END_IF

ELSE
	eMachineState									:=	E_SYSTEM_MachineState.POWERUP;

END_CASE

(*************************************write all system states to variables***********************)
stMachineState.bSystemPowerUp 						:=	(eMachineState=E_SYSTEM_MachineState.POWERUP);
IF stMachineState.bSystemPowerUp THEN 			sMachineState := aMachineState[1]; END_IF

stMachineState.bImmediateStopped 					:=	(eMachineState=E_SYSTEM_MachineState.IMMEDIATESTOPPED);
IF stMachineState.bImmediateStopped THEN 			sMachineState := aMachineState[2]; END_IF

stMachineState.bMachineInError 						:=	(eMachineState=E_SYSTEM_MachineState.MACHINEINERROR);
IF stMachineState.bMachineInError THEN 			sMachineState := aMachineState[3]; END_IF

stMachineState.bSystemInitialising 					:=	(eMachineState=E_SYSTEM_MachineState.INITIALISING);
IF stMachineState.bSystemInitialising THEN 			sMachineState := aMachineState[4]; END_IF

stMachineState.bManualMode 							:=	(eMachineState=E_SYSTEM_MachineState.MANUAL);
IF stMachineState.bManualMode THEN 			sMachineState := aMachineState[5]; END_IF

stMachineState.bSystemReadyToStart 					:=	(eMachineState=E_SYSTEM_MachineState.READYTOSTART);
IF stMachineState.bSystemReadyToStart THEN 			sMachineState := aMachineState[6]; END_IF

stMachineState.bSystemCycleStopping				:=	(eMachineState=E_SYSTEM_MachineState.STOPPING);
IF stMachineState.bSystemCycleStopping THEN 			sMachineState := aMachineState[7]; END_IF

stMachineState.bSystemRunning						:=	(eMachineState=E_SYSTEM_MachineState.RUNNING);
IF stMachineState.bSystemRunning THEN 			sMachineState := aMachineState[8]; END_IF

stMachineState.bMachineWaitingForProduct 			:=	(eMachineState=E_SYSTEM_MachineState.WAITINGFORPRODUCT);
IF stMachineState.bMachineWaitingForProduct THEN 			sMachineState := aMachineState[9]; END_IF

stMachineState.bTrackAndTraceDeactivated			:=	(eMachineState=E_SYSTEM_MachineState.PASSTHROUGHACTIVE);
IF stMachineState.bTrackAndTraceDeactivated THEN 			sMachineState := aMachineState[10]; END_IF

stMachineState.bMachineInConditionalRun 			:=	(eMachineState=E_SYSTEM_MachineState.CONDITIONALRUNNING);
IF stMachineState.bMachineInConditionalRun THEN 			sMachineState := aMachineState[11]; END_IF




IF sLastMachineState <> sMachineState THEN

	bMachineStateChanged	:= TRUE;
	sLastMachineState := sMachineState;
ELSE
	bMachineStateChanged	:= FALSE;
END_IF;

END_FUNCTION_BLOCK

// ---- POUs/METS/Common LIB/09_SYSTEM LIB/FB_SYSTEM_ProdMonitor.TcPOU
FUNCTION_BLOCK FB_SYSTEM_ProdMonitor
VAR_INPUT
	bEnable					: BOOL;
	stSystemTime				: TIMESTRUCT;
	(*bProductionChanged		: BOOL;*)
END_VAR
VAR_IN_OUT
	stPCMStatus				: ST_PCM_Status;	(* PCMstatus *)
	stCurrentStatisticNV		: ST_NOVRAM_METS_EventCounters;
	stCSVStoreTable			: ST_HMI_CSVStoreTable;

END_VAR
VAR_OUTPUT
	bProductionChanged			: BOOL;
	stLastProdOrder			: TIMESTRUCT;
END_VAR
VAR
	fbExecute					: R_TRIG;
END_VAR

(* shift manager disabled *)(* shift manager disabled *)
IF NOT bEnable  THEN

	(* clear outputs *)
	bProductionChanged := FALSE;
	MEMSET(ADR(stLastProdOrder), 16#00, SIZEOF(stLastProdOrder));

	RETURN;
END_IF

IF stCurrentStatisticNV.stEventStartDT.wYear = 0 AND stCurrentStatisticNV.stEventStartDT.wMonth = 0 THEN
	stCurrentStatisticNV.stEventStartDT := stSystemTime;
END_IF

(***************************Store current data to CSV structure for HMI******************************************)
fbExecute(CLK := stPCMStatus.bProductionChanged );

(* rising edge detected *)
IF fbExecute.Q = TRUE THEN

(*Blok przepisywania danych do  struct*)
	stCSVStoreTable.nShiftID 	:= 	0;
	stCSVStoreTable.sRSKU	:=	stCurrentStatisticNV.sRSKU;
	stCSVStoreTable.sProductionOrder	:=	stCurrentStatisticNV.sProductionOrder;

	stCSVStoreTable.stEventStartDT 	:= stCurrentStatisticNV.stEventStartDT;
	stCSVStoreTable.stEventEndDT 	:=  stSystemTime;

	MEMCPY(ADR(stCSVStoreTable.stMachineStateStatistic), ADR(stCurrentStatisticNV.stMachineStateStatistic), SIZEOF(stCSVStoreTable.stMachineStateStatistic));
	MEMCPY(ADR(stCSVStoreTable.aGeneralKPIStatistic), ADR(stCurrentStatisticNV.aGeneralKPIStatistic), SIZEOF(stCSVStoreTable.aGeneralKPIStatistic));
	MEMCPY(ADR(stCSVStoreTable.aAlarmsStatistic), ADR(stCurrentStatisticNV.aAlarmsStatistic), SIZEOF(stCSVStoreTable.aAlarmsStatistic));
	MEMCPY(ADR(stCSVStoreTable.aRejectCounters), ADR(stCurrentStatisticNV.aRejectCounters), SIZEOF(stCSVStoreTable.aRejectCounters));

	stCSVStoreTable.bDataStoredByHMI := TRUE;
	stLastProdOrder		:= stCSVStoreTable.stEventEndDT;

	MEMSET(ADR(stCurrentStatisticNV), 16#00, SIZEOF(stCurrentStatisticNV));

	stCurrentStatisticNV.sRSKU 				:= stPCMStatus.sRetailSKU;
	stCurrentStatisticNV.sProductionOrder  	:= stPCMStatus.sProductionOrder;

	stCurrentStatisticNV.stEventStartDT 	:= stSystemTime;

	bProductionChanged	:= TRUE;

ELSE
	bProductionChanged	:= FALSE;

END_IF

END_FUNCTION_BLOCK

// ---- POUs/METS/Common LIB/09_SYSTEM LIB/FB_SYSTEM_SearchBarcode.TcPOU
FUNCTION_BLOCK FB_SYSTEM_SearchBarcode
VAR_INPUT
	bExecute					: BOOL;
	bEnableInvalidSearch		: BOOL;
	bEnableCaseContentSearch	: BOOL;
	bEnablePackCodeRefeed		: BOOL ;
	bPackBarcode				: BOOL;
	bOuterIntermediate			: BOOL;
	bOuterBarcode				: BOOL;
	bCaseBarcode				: BOOL;
	sPackBarcode				: T_PACK_Barcode;
	sOuterIntermediateBarcode	: STRING(255);
	sOuterBarcode				: T_OUTER_Barcode;
	sCaseBarcode				: T_CASE_Barcode;
END_VAR
VAR_IN_OUT
	stCodeInfo_Pack			: ST_CodeInfo;
	stCodeInfo_Intermediate		: ST_CodeInfo;
	stCodeInfo_Outer			: ST_CodeInfo;

END_VAR
VAR_OUTPUT
	bDone					: BOOL;
	bBusy					: BOOL;
	bScanDone				: BOOL;
	sOutBarcode				: T_CASE_Barcode;
	sNewPackCodeRefeed		: T_PACK_Barcode;
END_VAR
VAR
	fbExRTrig 					: R_TRIG;
	fbExFTrig 					: F_TRIG;
	(*fbDecodeGS1				: FB_SCANNER_DecodeGS1;*)
	eCodeAIType				: E_CodeAIType;

	testString	 : STRING(255);

END_VAR

fbExRTrig(cLK:=bExecute);
fbExFTrig(cLK:=bExecute);

IF fbExRTrig.Q THEN
	bBusy := TRUE;
	bDone := FALSE;
	bScanDone := FALSE;
END_IF

IF fbExFTrig.Q THEN
	bBusy := FALSE;
	bDone := FALSE;
	bScanDone := FALSE;
END_IF

IF bBusy THEN

	IF NOT bEnableInvalidSearch AND bEnableCaseContentSearch AND NOT bEnablePackCodeRefeed THEN

		sNewPackCodeRefeed := '';

